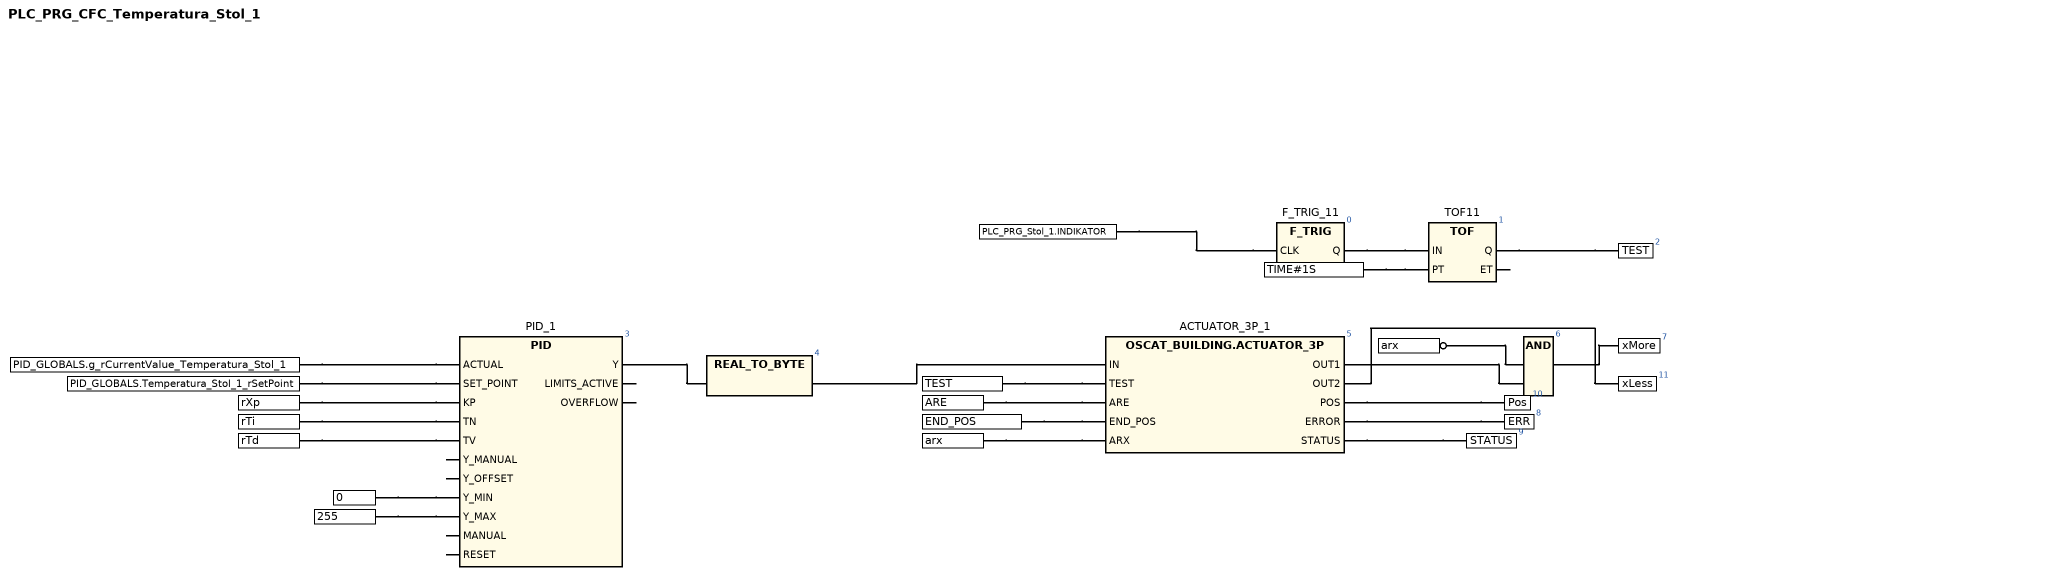
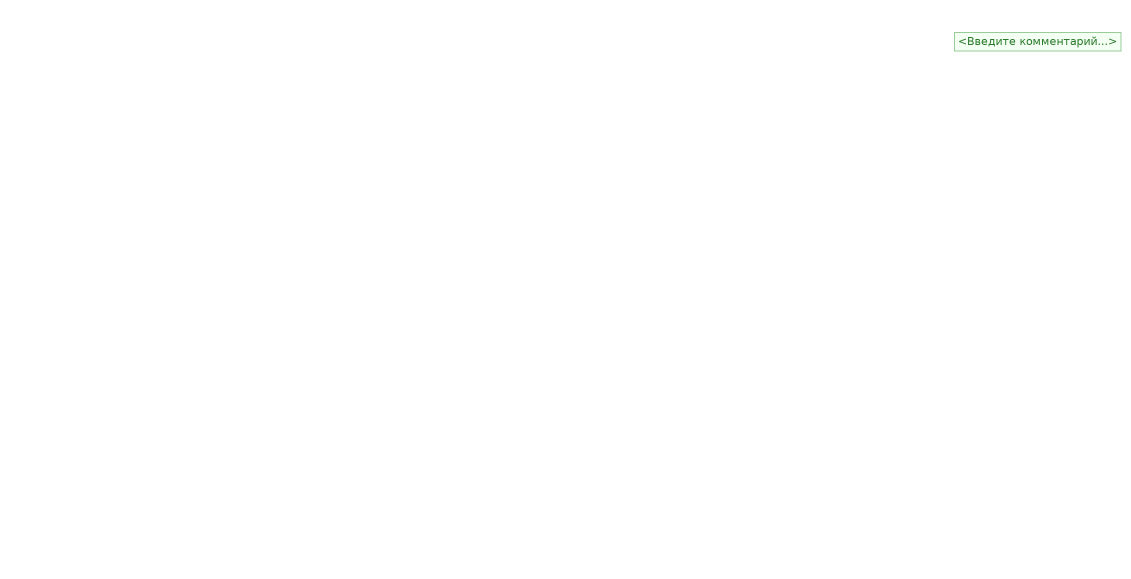
F_TRIG_11(CLK := PLC_PRG_Stol_1.INDIKATOR); // F_TRIG
TOF11(IN := F_TRIG_11.Q, PT := TIME#1S); // TOF
// <Введите комментарий...>
TEST := TOF11.Q;
PID_1(
    ACTUAL := PID_GLOBALS.g_rCurrentValue_Temperatura_Stol_1,
    SET_POINT := PID_GLOBALS.Temperatura_Stol_1_rSetPoint,
    KP := rXp,
    TN := rTi,
    TV := rTd,
    Y_MIN := 0,
    Y_MAX := 255); // PID
// parameter ACTUATOR_3P_1.SWITCH_AVAIL := FALSE
// parameter ACTUATOR_3P_1.T_DIAG := T#10d
// parameter ACTUATOR_3P_1.T_CAL := T#10m
// parameter ACTUATOR_3P_1.T_EXT := T#10s
// parameter ACTUATOR_3P_1.T_RUN := PLC_PRG_CFC_Temperatura_Stol_1.Time_RUN
ACTUATOR_3P_1(IN := REAL_TO_BYTE(PID_1.Y), TEST := TEST, ARE := ARE, END_POS := END_POS, ARX := arx); // OSCAT_BUILDING.ACTUATOR_3P
xMore := NOT arx AND ACTUATOR_3P_1.OUT1;
ERR := ACTUATOR_3P_1.ERROR;
STATUS := ACTUATOR_3P_1.STATUS;
Pos := ACTUATOR_3P_1.POS;
xLess := ACTUATOR_3P_1.OUT2;

END_PROGRAM

// Device/Application/CFC_Temperatura_PID/PLC_PRG_CFC_Temperatura_Stol_3
PROGRAM PLC_PRG_CFC_Temperatura_Stol_3
VAR
	ACTUATOR_3P_1:		OSCAT_BUILDING.ACTUATOR_3P;
	PID_1: 				PID;						// ФБ ПИД
	arx: 				BOOL;
	xMore:				BOOL;						// Сигнал открытия
	xLess: 				BOOL;						// Сигнал на закрытие	
	TEST: 				BOOL;						// Переменная запускающая тестирование ФБ ACTUATOR_3P
	Pos: 				BYTE;						// Переменная принимающая позицию 3-х ходового клапана виртуальную
	
	ARE: BOOL;
	END_POS: BOOL;
	ERR: BOOL;
	STATUS: BYTE;
	F_TRIG_21: F_TRIG;
	TOF21: TOF;
END_VAR

VAR RETAIN
	rXp: 									REAL:=2;					// Полоса пропускания (100/Кр)
	rTi: 									REAL:=25;					// Постоянная времени интегрирования
	rTd: 									REAL:=0.01;					// Постоянная времени дифференцирования
	Time_RUN:								TIME:=T#120S;				// Время хода 3-х ходового клапана
END_VAR

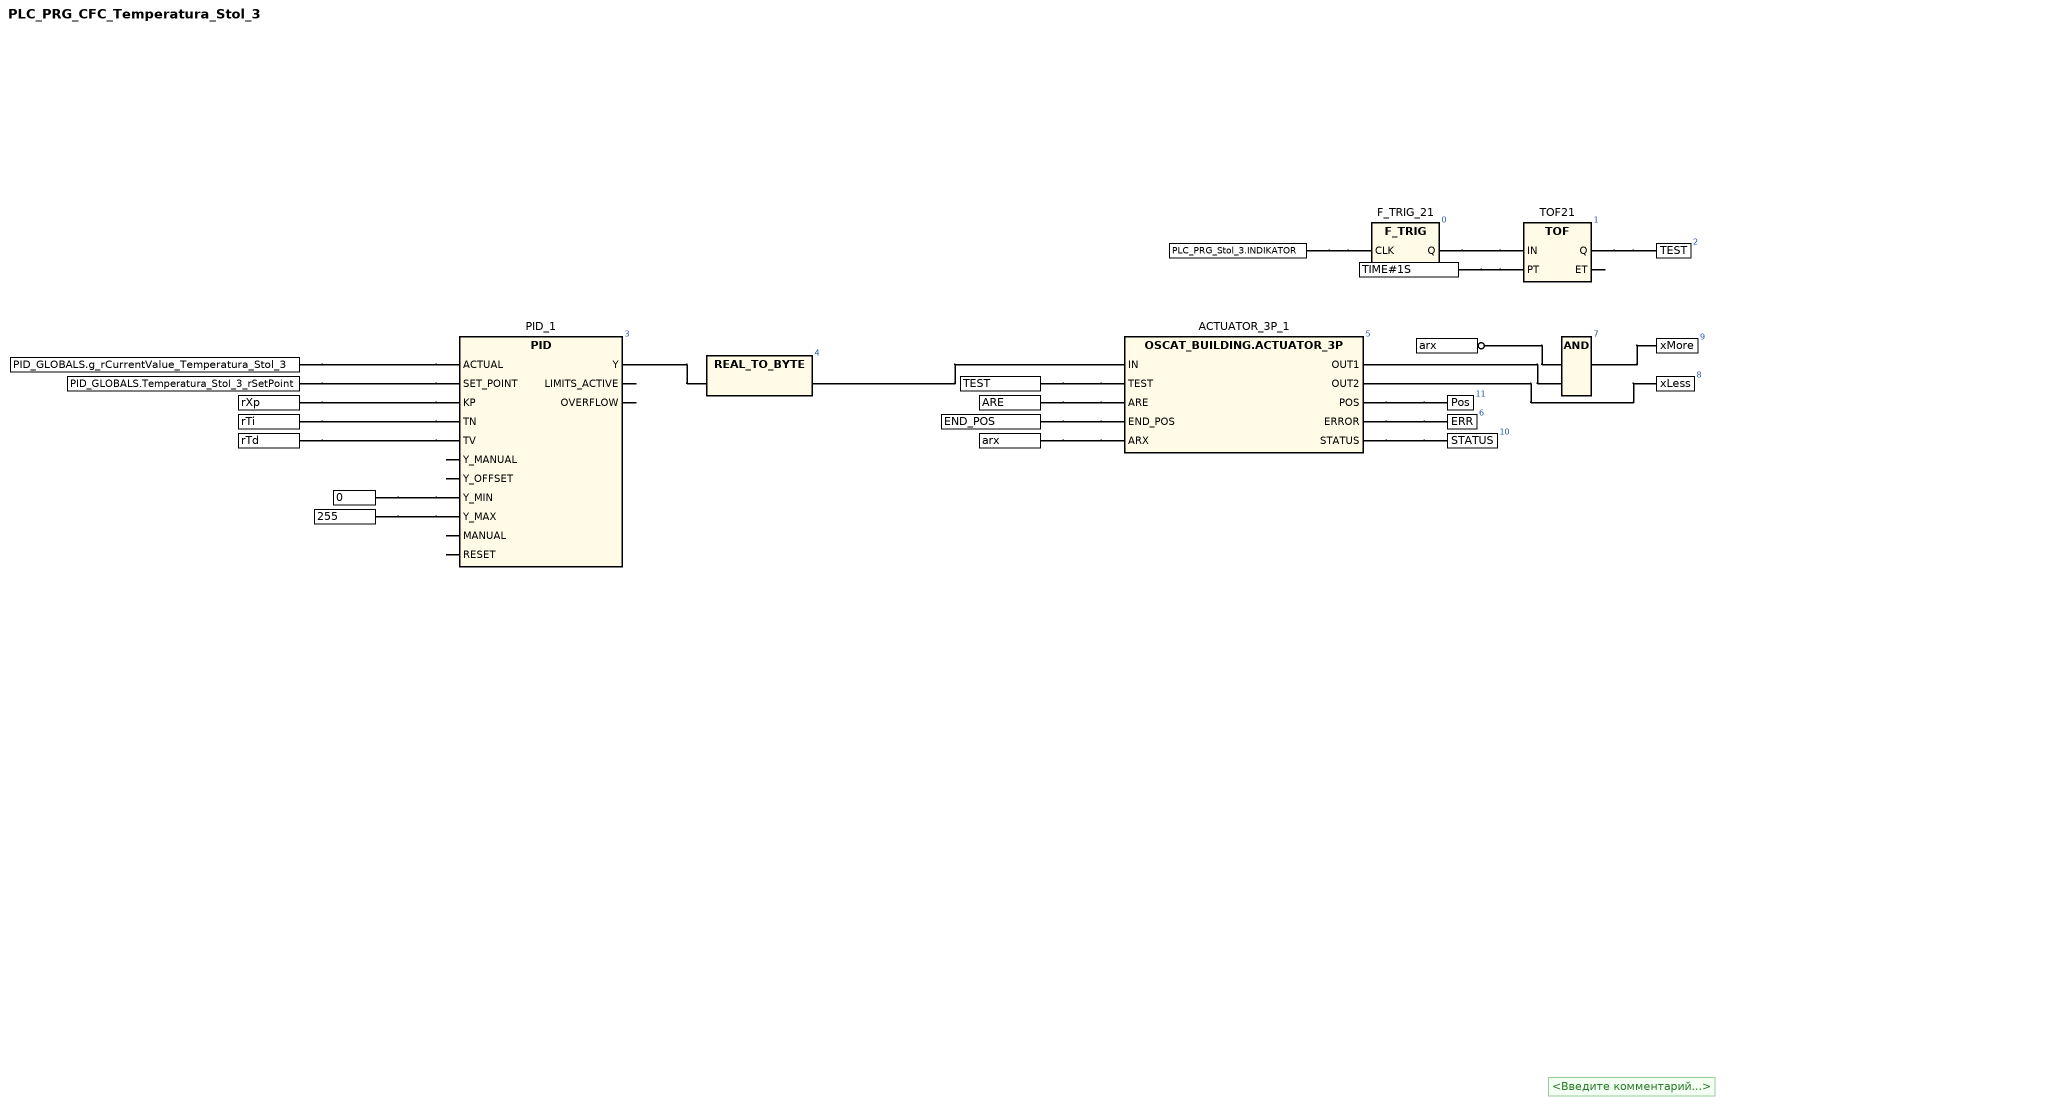
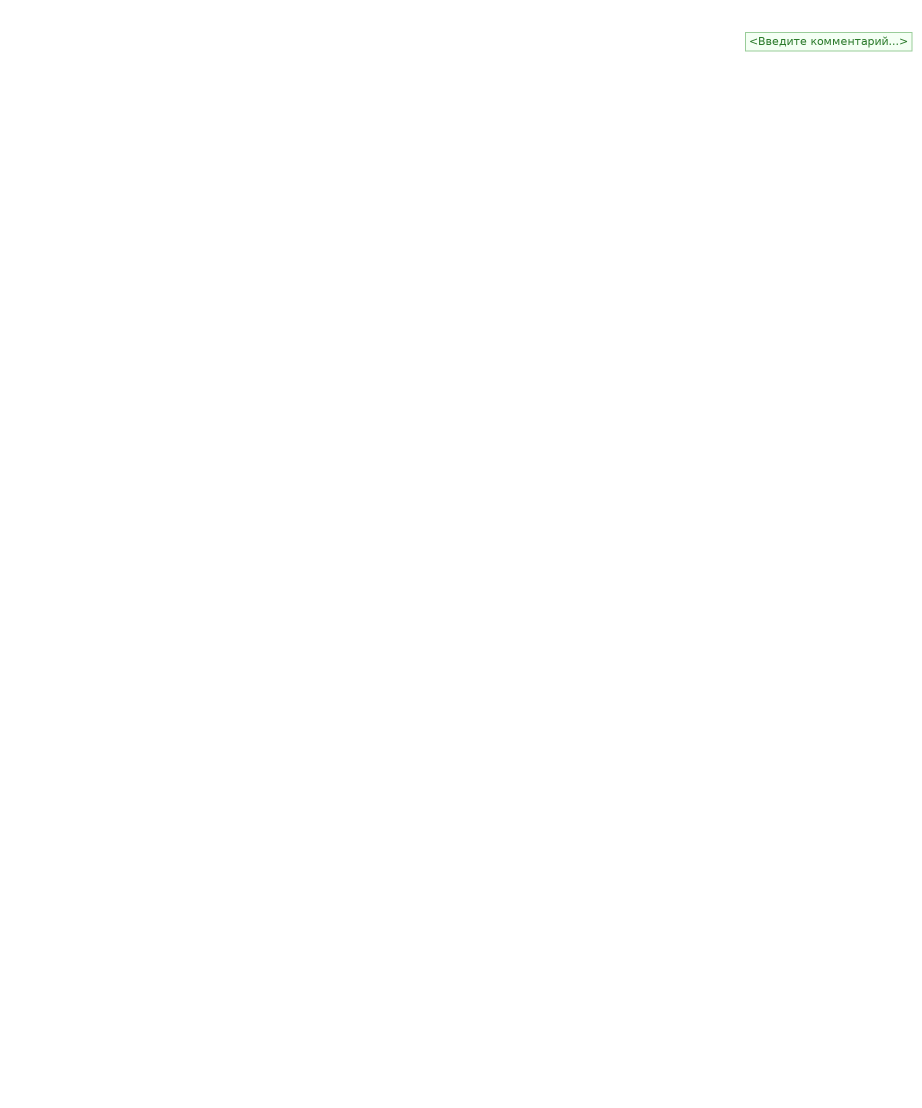
F_TRIG_21(CLK := PLC_PRG_Stol_3.INDIKATOR); // F_TRIG
TOF21(IN := F_TRIG_21.Q, PT := TIME#1S); // TOF
// <Введите комментарий...>
TEST := TOF21.Q;
PID_1(
    ACTUAL := PID_GLOBALS.g_rCurrentValue_Temperatura_Stol_3,
    SET_POINT := PID_GLOBALS.Temperatura_Stol_3_rSetPoint,
    KP := rXp,
    TN := rTi,
    TV := rTd,
    Y_MIN := 0,
    Y_MAX := 255); // PID
// parameter ACTUATOR_3P_1.SWITCH_AVAIL := FALSE
// parameter ACTUATOR_3P_1.T_DIAG := T#10d
// parameter ACTUATOR_3P_1.T_CAL := T#10m
// parameter ACTUATOR_3P_1.T_EXT := T#10s
// parameter ACTUATOR_3P_1.T_RUN := PLC_PRG_CFC_Temperatura_Stol_3.Time_RUN
ACTUATOR_3P_1(IN := REAL_TO_BYTE(PID_1.Y), TEST := TEST, ARE := ARE, END_POS := END_POS, ARX := arx); // OSCAT_BUILDING.ACTUATOR_3P
ERR := ACTUATOR_3P_1.ERROR;
xLess := ACTUATOR_3P_1.OUT2;
xMore := NOT arx AND ACTUATOR_3P_1.OUT1;
// <Введите комментарий...>
STATUS := ACTUATOR_3P_1.STATUS;
Pos := ACTUATOR_3P_1.POS;

END_PROGRAM

// Device/Application/CFC_Temperatura_PID/PLC_PRG_CFC_Temperatura_Stol_4
PROGRAM PLC_PRG_CFC_Temperatura_Stol_4
VAR
	ACTUATOR_3P_1:		OSCAT_BUILDING.ACTUATOR_3P;
	PID_1: 				PID;						// ФБ ПИД
	arx: 				BOOL;
	xMore:				BOOL;						// Сигнал открытия
	xLess: 				BOOL;						// Сигнал на закрытие
	
	TEST: 				BOOL;						// Переменная запускающая тестирование ФБ ACTUATOR_3P
	Pos: 				BYTE;						// Переменная принимающая позицию 3-х ходового клапана виртуальную
	
	ARE: BOOL;
	END_POS: BOOL;
	ERR: BOOL;
	STATUS: BYTE;
	F_TRIG_11: F_TRIG;
	TOF11: TOF;
END_VAR

VAR RETAIN	
	rXp: 									REAL:=2;					// Полоса пропускания (100/Кр)
	rTi: 									REAL:=25;					// Постоянная времени интегрирования
	rTd: 									REAL:=0.01;					// Постоянная времени дифференцирования
	Time_RUN:								TIME:=T#120S;				// Время хода 3-х ходового клапана
END_VAR

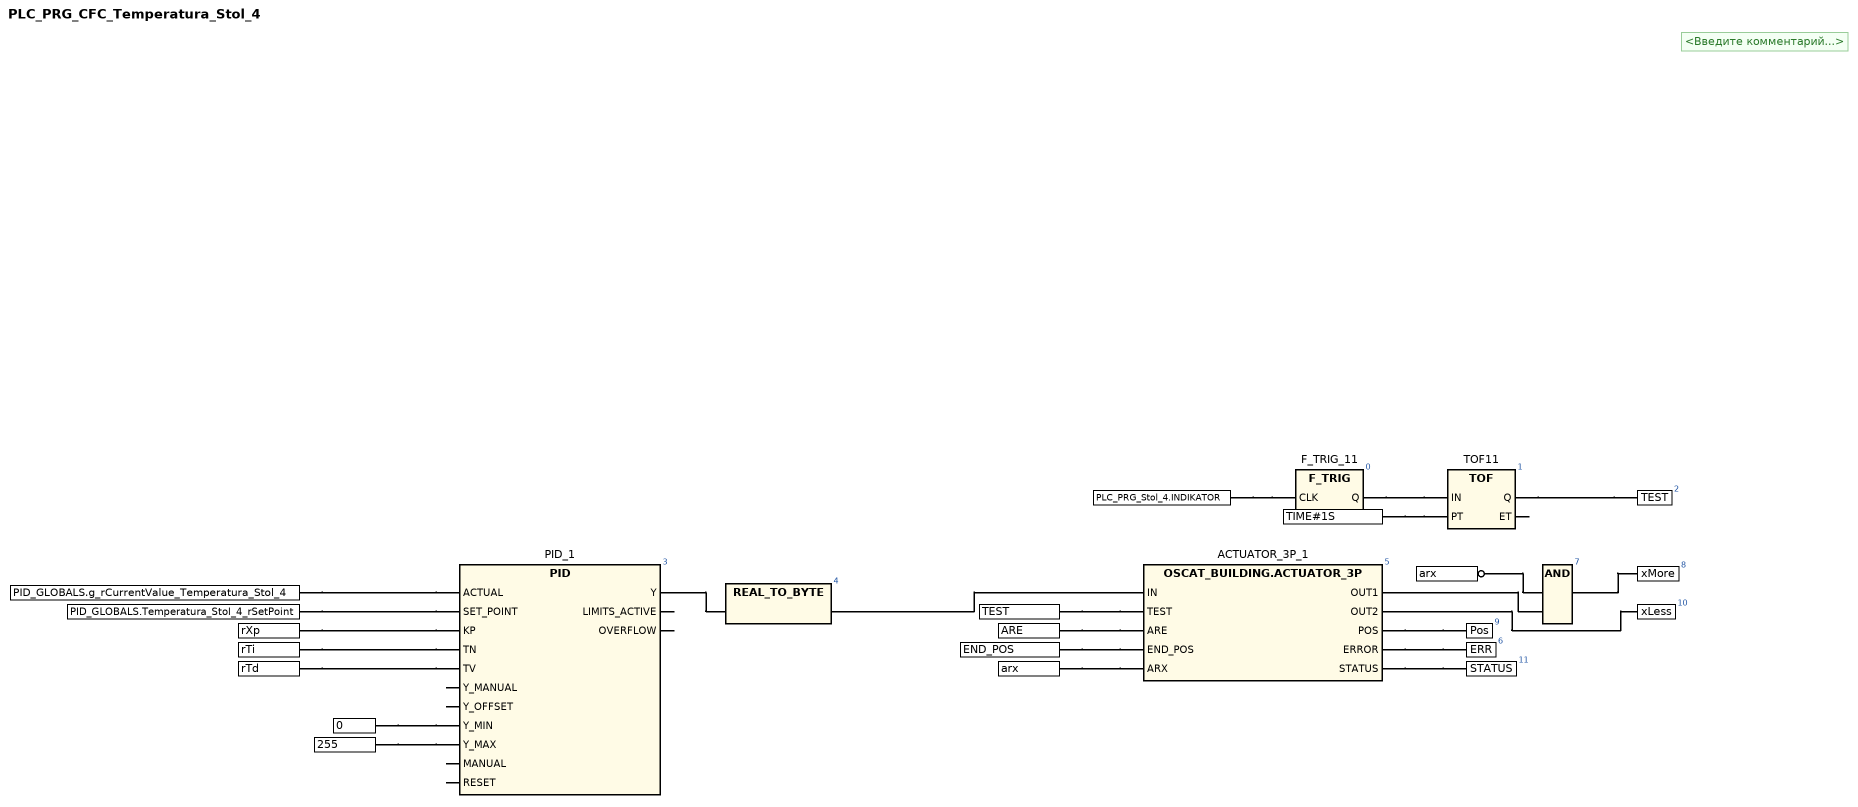
F_TRIG_11(CLK := PLC_PRG_Stol_4.INDIKATOR); // F_TRIG
TOF11(IN := F_TRIG_11.Q, PT := TIME#1S); // TOF
// <Введите комментарий...>
TEST := TOF11.Q;
PID_1(
    ACTUAL := PID_GLOBALS.g_rCurrentValue_Temperatura_Stol_4,
    SET_POINT := PID_GLOBALS.Temperatura_Stol_4_rSetPoint,
    KP := rXp,
    TN := rTi,
    TV := rTd,
    Y_MIN := 0,
    Y_MAX := 255); // PID
// parameter ACTUATOR_3P_1.SWITCH_AVAIL := FALSE
// parameter ACTUATOR_3P_1.T_DIAG := T#10d
// parameter ACTUATOR_3P_1.T_CAL := T#10m
// parameter ACTUATOR_3P_1.T_EXT := T#10s
// parameter ACTUATOR_3P_1.T_RUN := PLC_PRG_CFC_Temperatura_Stol_4.Time_RUN
ACTUATOR_3P_1(IN := REAL_TO_BYTE(PID_1.Y), TEST := TEST, ARE := ARE, END_POS := END_POS, ARX := arx); // OSCAT_BUILDING.ACTUATOR_3P
ERR := ACTUATOR_3P_1.ERROR;
xMore := NOT arx AND ACTUATOR_3P_1.OUT1;
Pos := ACTUATOR_3P_1.POS;
xLess := ACTUATOR_3P_1.OUT2;
STATUS := ACTUATOR_3P_1.STATUS;

END_PROGRAM

// Device/Application/archive/PLC_PRG_archive
PROGRAM PLC_PRG_archive
VAR
	//проверка работы архива
	//xArchEnable:				BOOL;								// бит управления архиватором
	xArchError_1:				OwenArchiverErrors.ARCHIVE_ERROR;	// код ошибки
	wsArchError_1:				WSTRING;							// сообщение об ошибке
	xArchStatus_1:				BOOL;								// статус архиватора (TRUE - запущен, FALSE - остановлен)

	// 3 и 4 стол
	xArchError_3_4:				OwenArchiverErrors.ARCHIVE_ERROR;	// код ошибки
	wsArchError_3_4:			WSTRING;							// сообщение об ошибке
	xArchStatus_3_4:			BOOL;								// статус архиватора (TRUE - запущен, FALSE - остановлен)
	
	La_rat:						BOOL;								// памяти осталось меньше 2 ГБ
	rat:						REAL;								// конвертация wstring в sint
	
	Name:						STRING;								// Имя человека активного сейчас
	
	// информация о накопителе
	xDriveInfo:					BOOL;								// режим сбора данных (TRUE - вкл.)
	
	stPlcMemory:				DriveInfo;							// структура параметров памяти контроллера
	stUsbMemory:				DriveInfo;							// структура параметров памяти USB-накопителя 
	
	fbUsbUnmountTimeout:		TON;								// таймер сброса флага "USB отмонтирован"
	
	xArchError_3_4_1:			OwenArchiverErrors.ARCHIVE_ERROR;	// статус архиватора (TRUE - запущен, FALSE - остановлен)
	warning_2:					BOOL;								// Ошибка остановлена архивация на флешку	
	warning_3:					BOOL;								// Ошибка "Неверный путь ведения архива"
	warning_4:					BOOL;								// Ошибка "Ошибка создания структуры директорий"
	warning_5:					BOOL;								// Ошибка "Ошибка удаления файла"
	warning_6:					BOOL;								// Ошибка "Ошибка переименования файла"
	warning_7:					BOOL;								// Ошибка "Некорректный буфер записи"
	warning_8:					BOOL;								// Ошибка "Некорректный размер буфера записи"
	warning_9:					BOOL;								// Ошибка "Не задан список переменных"
	warning_10:					BOOL;								// Ошибка "Список переменных пуст"
	warning_11:					BOOL;								// Ошибка "Ошибка записи"
	warning_12:					BOOL;								// Ошибка "Ошибка создания заголовка файла"
	warning_13:					BOOL;								// Ошибка "Ошибка буфер переполнен"
	
	
	x1:							BOOL;								// Отображение измененинй на 1 столе
	y1:							BOOL;								// Отображение измененинй на 3 столе
	z1:							BOOL;								// Отображение измененинй на 4 столе
	
END_VAR

// конвертируем код ошибки архиватора в строку
wsArchError_1 := OwenArchiverErrors.ARCHIVE_ERROR_TO_WSTRING(xArchError_1);

// конвертируем код ошибки архиватора в строку
wsArchError_3_4 := OwenArchiverErrors.ARCHIVE_ERROR_TO_WSTRING(xArchError_3_4);

act01_DriveInfo();			// сбор информации о памяти накомпителя и ПЛК

rat := WSTRING_TO_SINT(stUsbMemory.wsFreeSize);

IF rat > 2  THEN				// поменять цифру 2 на 4 когда придёт флешка
	La_rat  := TRUE;			// надо почистить флешку на термостолах
END_IF

// Проверка записи архива на флешку
IF xArchStatus_1 = TRUE OR xArchStatus_3_4 = TRUE THEN
	warning_2 := TRUE;
ELSE
	warning_2 := FALSE;
END_IF

Name := TO_STRING(VisuElems.CurrentFullUserName);


// Определение последней ошибки архивации
IF xArchError_3_4_1 = ARCHIVE_ERROR.INCORRECT_ARCHIVE_PATH THEN
	warning_3 := TRUE;
	warning_4 := FALSE;
	warning_5 := FALSE;
	warning_6 := FALSE;
	warning_7 := FALSE;
	warning_8 := FALSE;
	warning_9 := FALSE;
	warning_10 := FALSE;
	warning_11 := FALSE;
	warning_12 := FALSE;
	warning_13 := FALSE;
	ELSIF xArchError_3_4_1 = ARCHIVE_ERROR.CREATE_FOLDER_STRUCTURE_ERROR THEN
	warning_4 := TRUE;
	warning_3 := FALSE;
	warning_5 := FALSE;
	warning_6 := FALSE;
	warning_7 := FALSE;
	warning_8 := FALSE;
	warning_9 := FALSE;
	warning_10 := FALSE;
	warning_11 := FALSE;
	warning_12 := FALSE;
	warning_13 := FALSE;
	ELSIF xArchError_3_4_1 = ARCHIVE_ERROR.DELETE_FILE_ERROR THEN
	warning_5 := TRUE;
	warning_3 := FALSE;
	warning_4 := FALSE;
	warning_6 := FALSE;
	warning_7 := FALSE;
	warning_8 := FALSE;
	warning_9 := FALSE;
	warning_10 := FALSE;
	warning_11 := FALSE;
	warning_12 := FALSE;
	warning_13 := FALSE;
	ELSIF xArchError_3_4_1 = ARCHIVE_ERROR.RENAME_FILE_ERROR THEN
	warning_3 := FALSE;
	warning_4 := FALSE;
	warning_5 := FALSE;
	warning_6 := TRUE;
	warning_7 := FALSE;
	warning_8 := FALSE;
	warning_9 := FALSE;
	warning_10 := FALSE;
	warning_11 := FALSE;
	warning_12 := FALSE;
	warning_13 := FALSE;
	ELSIF xArchError_3_4_1 = ARCHIVE_ERROR.INCORRECT_WRITER_BUFFER THEN
	warning_3 := FALSE;
	warning_4 := FALSE;
	warning_5 := FALSE;
	warning_6 := FALSE;
	warning_7 := TRUE;
	warning_8 := FALSE;
	warning_9 := FALSE;
	warning_10 := FALSE;
	warning_11 := FALSE;
	warning_12 := FALSE;
	warning_13 := FALSE;
	ELSIF xArchError_3_4_1 = ARCHIVE_ERROR.INCORRECT_WRITER_BUFFER_SIZE THEN
	warning_3 := FALSE;
	warning_4 := FALSE;
	warning_5 := FALSE;
	warning_6 := FALSE;
	warning_7 := FALSE;
	warning_8 := TRUE;
	warning_9 := FALSE;
	warning_10 := FALSE;
	warning_11 := FALSE;
	warning_12 := FALSE;
	warning_13 := FALSE;
	ELSIF xArchError_3_4_1 = ARCHIVE_ERROR.VARIABLE_LIST_NOT_SPECIFIED THEN
	warning_3 := FALSE;
	warning_4 := FALSE;
	warning_5 := FALSE;
	warning_6 := FALSE;
	warning_7 := FALSE;
	warning_8 := FALSE;
	warning_9 := TRUE;
	warning_10 := FALSE;
	warning_11 := FALSE;
	warning_12 := FALSE;
	warning_13 := FALSE;
	ELSIF xArchError_3_4_1 = ARCHIVE_ERROR.VARIABLE_LIST_IS_EMPTY THEN
	warning_3 := FALSE;
	warning_4 := FALSE;
	warning_5 := FALSE;
	warning_6 := FALSE;
	warning_7 := FALSE;
	warning_8 := FALSE;
	warning_9 := FALSE;
	warning_10 := TRUE;
	warning_11 := FALSE;
	warning_12 := FALSE;
	warning_13 := FALSE;
	ELSIF xArchError_3_4_1 = ARCHIVE_ERROR.WRITE_ERROR THEN
	warning_3 := FALSE;
	warning_4 := FALSE;
	warning_5 := FALSE;
	warning_6 := FALSE;
	warning_7 := FALSE;
	warning_8 := FALSE;
	warning_9 := FALSE;
	warning_10 := FALSE;
	warning_11 := TRUE;
	warning_12 := FALSE;
	warning_13 := FALSE;
	ELSIF xArchError_3_4_1 = ARCHIVE_ERROR.CREATE_HEADER_ERROR THEN
	warning_3 := FALSE;
	warning_4 := FALSE;
	warning_5 := FALSE;
	warning_6 := FALSE;
	warning_7 := FALSE;
	warning_8 := FALSE;
	warning_9 := FALSE;
	warning_10 := FALSE;
	warning_11 := FALSE;
	warning_12 := TRUE;
	warning_13 := FALSE;
	ELSIF xArchError_3_4_1 = ARCHIVE_ERROR.WRITE_BUFFER_OVERFLOW THEN
	warning_3 := FALSE;
	warning_4 := FALSE;
	warning_5 := FALSE;
	warning_6 := FALSE;
	warning_7 := FALSE;
	warning_8 := FALSE;
	warning_9 := FALSE;
	warning_10 := FALSE;
	warning_11 := FALSE;
	warning_12 := FALSE;
	warning_13 := TRUE;
	ELSE
	warning_3 := FALSE;
	warning_4 := FALSE;
	warning_5 := FALSE;
	warning_6 := FALSE;
	warning_7 := FALSE;
	warning_8 := FALSE;
	warning_9 := FALSE;
	warning_10 := FALSE;
	warning_11 := FALSE;
	warning_12 := FALSE;
	warning_13 := FALSE;
END_IF

ACTION act01_DriveInfo:
// преобразование размеров полной/занятой/свободной памяти в форматированную строку

stPlcMemory.wsFullSize 		:= BYTE_SIZE_TO_WSTRING(stPlcMemory.uleFullSize);
stPlcMemory.wsUsedSize 		:= BYTE_SIZE_TO_WSTRING(stPlcMemory.uleUsedSize);
stPlcMemory.wsFreeSize 		:= BYTE_SIZE_TO_WSTRING(stPlcMemory.uleFreeSize);

stUsbMemory.wsFullSize 		:= BYTE_SIZE_TO_WSTRING(stUsbMemory.uleFullSize);
stUsbMemory.wsUsedSize 		:= BYTE_SIZE_TO_WSTRING(stUsbMemory.uleUsedSize);
stUsbMemory.wsFreeSize 		:= BYTE_SIZE_TO_WSTRING(stUsbMemory.uleFreeSize);

// сброс флагов "устройство отмонтировано" через 5 секунд после отмонтирования устройства
fbUsbUnmountTimeout(IN:=stUsbMemory.xUnmountDone, PT:=T#5S);

IF fbUsbUnmountTimeout.Q THEN
	stUsbMemory.xUnmount:=FALSE;
END_IF
END_ACTION

END_PROGRAM

// Device/Application/archive/BYTE_SIZE_TO_WSTRING
// функция преобразования числа байт в форматированную строку
FUNCTION BYTE_SIZE_TO_WSTRING : WSTRING
VAR_INPUT
	uliByteSize: 				ULINT; 				// число байт
END_VAR
VAR CONSTANT
	c_uliBytePerKilobyte: 		ULINT := 1024; 		// число байт в килобайте
	c_uliKilobytePerMegabyte: 	ULINT := 1024 * c_uliBytePerKilobyte;
	c_uliMegabytePerGigabyte: 	ULINT := 1024 * c_uliKilobytePerMegabyte;
END_VAR
VAR
	rByteSize: 					REAL; 				// промежуточная переменная
END_VAR

CASE uliByteSize OF
	

	0 ..(c_uliBytePerKilobyte - 1):
			BYTE_SIZE_TO_WSTRING := WCONCAT(ULINT_TO_WSTRING(uliByteSize), " Байт");

	c_uliBytePerKilobyte ..(c_uliKilobytePerMegabyte - 1):
			rByteSize := ULINT_TO_REAL(uliByteSize) / ULINT_TO_REAL(c_uliBytePerKilobyte);
			BYTE_SIZE_TO_WSTRING := WCONCAT(REAL_TO_FWSTRING(rByteSize, 2), " Кбайт");

	c_uliKilobytePerMegabyte ..(c_uliMegabytePerGigabyte - 1):
			rByteSize := ULINT_TO_REAL(uliByteSize) / ULINT_TO_REAL(c_uliKilobytePerMegabyte);
			BYTE_SIZE_TO_WSTRING := WCONCAT(REAL_TO_FWSTRING(rByteSize, 2), " Мбайт");

	c_uliMegabytePerGigabyte ..(32 * c_uliMegabytePerGigabyte):
			rByteSize := ULINT_TO_REAL(uliByteSize) / ULINT_TO_REAL(c_uliMegabytePerGigabyte);
			BYTE_SIZE_TO_WSTRING := WCONCAT(REAL_TO_FWSTRING(rByteSize, 2), " Гбайт");
			
END_CASE

END_FUNCTION

// Device/Application/archive/REAL_TO_FWSTRING
// функция конвертирует значение типа REAL в строку с n знаков после запятой
FUNCTION REAL_TO_FWSTRING : WSTRING

VAR_INPUT
	rVar: 			REAL; 		// входное значение
	usiPrecision: 	USINT; 		// нужное кол-во знаков после запятой
END_VAR
VAR
	uliVar: 		ULINT; 		// промежуточная переменная
	lrVar: 			LREAL; 		// промежуточная переменная
END_VAR



uliVar := LREAL_TO_ULINT( (rVar)*EXPT(10, usiPrecision) );
lrVar := LINT_TO_LREAL(uliVar) / EXPT(10, usiPrecision);
REAL_TO_FWSTRING := LREAL_TO_WSTRING(lrVar);

END_FUNCTION

// Device/Application/Connection
PROGRAM Connection
VAR
	// Модуль расширения MK210_311_Stol_1_2
	sName_MK210_311_Stol_1_2:					STRING;						// Имя модуля, считанное с модуля
	sProjectName_MK210_311_Stol_1_2:			STRING;						// Имя модуля в дереве проекта
	abyIP_MK210_311_Stol_1_2:					ARRAY [0..3] OF BYTE;		// IP-адрес в дереве проекта
	sFactoryNumber_MK210_311_Stol_1_2:			STRING;						// заводской номер модуля
	udiErrorsCount_MK210_311_Stol_1_2:			UDINT;						// Число ошибок связи с модулем с последней загрузки контроллера
	eLastError_MK210_311_Stol_1_2: 				MB_ERRORCODES;				// код последней ошибки
	ePollState_MK210_311_Stol_1_2:				MODULE_STATE;				// состояние опроса
	
	// Модуль расширения MV210_212_Stol_1_2
	sName_MV210_212_Stol_1_2:					STRING;						// Имя модуля, считанное с модуля
	sProjectName_MV210_212_Stol_1_2:			STRING;						// Имя модуля в дереве проекта
	abyIP_MV210_212_Stol_1_2:					ARRAY [0..3] OF BYTE;		// IP-адрес в дереве проекта
	sFactoryNumber_MV210_212_Stol_1_2:			STRING;						// заводской номер модуля
	udiErrorsCount_MV210_212_Stol_1_2:			UDINT;						// Число ошибок связи с модулем с последней загрузки контроллера
	eLastError_MV210_212_Stol_1_2: 				MB_ERRORCODES;				// код последней ошибки
	ePollState_MV210_212_Stol_1_2:				MODULE_STATE;				// состояние опроса
	
	// Модуль расширения MV210_101_Stol_1_2
	sName_MV210_101_Stol_1_2:					STRING;						// Имя модуля, считанное с модуля
	sProjectName_MV210_101_Stol_1_2:			STRING;						// Имя модуля в дереве проекта
	abyIP_MV210_101_Stol_1_2:					ARRAY [0..3] OF BYTE;		// IP-адрес в дереве проекта
	sFactoryNumber_MV210_101_Stol_1_2:			STRING;						// заводской номер модуля
	udiErrorsCount_MV210_101_Stol_1_2:			UDINT;						// Число ошибок связи с модулем с последней загрузки контроллера
	eLastError_MV210_101_Stol_1_2: 				MB_ERRORCODES;				// код последней ошибки
	ePollState_MV210_101_Stol_1_2:				MODULE_STATE;				// состояние опроса
	
	// Модуль расширения MK210_311_Stol_3_4
	sName_MK210_311_Stol_3_4:					STRING;						// Имя модуля, считанное с модуля
	sProjectName_MK210_311_Stol_3_4:			STRING;						// Имя модуля в дереве проекта
	abyIP_MK210_311_Stol_3_4:					ARRAY [0..3] OF BYTE;		// IP-адрес в дереве проекта
	sFactoryNumber_MK210_311_Stol_3_4:			STRING;						// заводской номер модуля
	udiErrorsCount_MK210_311_Stol_3_4:			UDINT;						// Число ошибок связи с модулем с последней загрузки контроллера
	eLastError_MK210_311_Stol_3_4: 				MB_ERRORCODES;				// код последней ошибки
	ePollState_MK210_311_Stol_3_4:				MODULE_STATE;				// состояние опроса
	
	// Модуль расширения MV210_212_Stol_3_4
	sName_MV210_212_Stol_3_4:					STRING;						// Имя модуля, считанное с модуля
	sProjectName_MV210_212_Stol_3_4:			STRING;						// Имя модуля в дереве проекта
	abyIP_MV210_212_Stol_3_4:					ARRAY [0..3] OF BYTE;		// IP-адрес в дереве проекта
	sFactoryNumber_MV210_212_Stol_3_4:			STRING;						// заводской номер модуля
	udiErrorsCount_MV210_212_Stol_3_4:			UDINT;						// Число ошибок связи с модулем с последней загрузки контроллера
	eLastError_MV210_212_Stol_3_4: 				MB_ERRORCODES;				// код последней ошибки
	ePollState_MV210_212_Stol_3_4:				MODULE_STATE;				// состояние опроса
	
	// Модуль расширения MV210_101_Stol_3_4
	sName_MV210_101_Stol_3_4:					STRING;						// Имя модуля, считанное с модуля
	sProjectName_MV210_101_Stol_3_4:			STRING;						// Имя модуля в дереве проекта
	abyIP_MV210_101_Stol_3_4:					ARRAY [0..3] OF BYTE;		// IP-адрес в дереве проекта
	sFactoryNumber_MV210_101_Stol_3_4:			STRING;						// Pаводской номер модуля
	udiErrorsCount_MV210_101_Stol_3_4:			UDINT;						// Число ошибок связи с модулем с последней загрузки контроллера
	eLastError_MV210_101_Stol_3_4: 				MB_ERRORCODES;				// Rод последней ошибки
	ePollState_MV210_101_Stol_3_4:				MODULE_STATE;				// Cостояние опроса
		
	warning:									BOOL;						// Ошибка модулей расширения 1 стола
	warning_1:									BOOL;						// Ошибка модулей расширения 3 и 4 столов
END_VAR

// Модуль расширения MK210_311_Stol_1_2
sName_MK210_311_Stol_1_2				:=  MK210_311_Stol_1_2_OwenDriver.Name;
sProjectName_MK210_311_Stol_1_2			:=	MK210_311_Stol_1_2_OwenDriver.ProjectName;
abyIP_MK210_311_Stol_1_2				:=	MK210_311_Stol_1_2_OwenDriver.Ip;
sFactoryNumber_MK210_311_Stol_1_2 		:=	MK210_311_Stol_1_2_OwenDriver.FactoryNumber;
udiErrorsCount_MK210_311_Stol_1_2		:=	MK210_311_Stol_1_2_OwenDriver.ErrorsCount;
eLastError_MK210_311_Stol_1_2 			:=	MK210_311_Stol_1_2_OwenDriver.LastError;
ePollState_MK210_311_Stol_1_2			:=	MK210_311_Stol_1_2_OwenDriver.PollState;

// Модуль расширения MV210_212_Stol_1_2
sName_MV210_212_Stol_1_2				:=  MV210_212_Stol_1_2_OwenDriver.Name;
sProjectName_MV210_212_Stol_1_2			:=	MV210_212_Stol_1_2_OwenDriver.ProjectName;
abyIP_MV210_212_Stol_1_2				:=	MV210_212_Stol_1_2_OwenDriver.Ip;
sFactoryNumber_MV210_212_Stol_1_2 		:=	MV210_212_Stol_1_2_OwenDriver.FactoryNumber;
udiErrorsCount_MV210_212_Stol_1_2		:=	MV210_212_Stol_1_2_OwenDriver.ErrorsCount;
eLastError_MV210_212_Stol_1_2 			:=	MV210_212_Stol_1_2_OwenDriver.LastError;
ePollState_MV210_212_Stol_1_2			:=	MV210_212_Stol_1_2_OwenDriver.PollState;

// Модуль расширения MV210_101_Stol_1_2
sName_MV210_101_Stol_1_2				:=  MV210_101_Stol_1_2_OwenDriver.Name;
sProjectName_MV210_101_Stol_1_2			:=	MV210_101_Stol_1_2_OwenDriver.ProjectName;
abyIP_MV210_101_Stol_1_2				:=	MV210_101_Stol_1_2_OwenDriver.Ip;
sFactoryNumber_MV210_101_Stol_1_2	 	:=	MV210_101_Stol_1_2_OwenDriver.FactoryNumber;
udiErrorsCount_MV210_101_Stol_1_2		:=	MV210_101_Stol_1_2_OwenDriver.ErrorsCount;
eLastError_MV210_101_Stol_1_2 			:=	MV210_101_Stol_1_2_OwenDriver.LastError;
ePollState_MV210_101_Stol_1_2			:=	MV210_101_Stol_1_2_OwenDriver.PollState;

// Модуль расширения MK210_311_Stol_3_4
sName_MK210_311_Stol_3_4				:=  MK210_311_Stol_3_4_OwenDriver.Name;
sProjectName_MK210_311_Stol_3_4			:=	MK210_311_Stol_3_4_OwenDriver.ProjectName;
abyIP_MK210_311_Stol_3_4				:=	MK210_311_Stol_3_4_OwenDriver.Ip;
sFactoryNumber_MK210_311_Stol_3_4 		:=	MK210_311_Stol_3_4_OwenDriver.FactoryNumber;
udiErrorsCount_MK210_311_Stol_3_4		:=	MK210_311_Stol_3_4_OwenDriver.ErrorsCount;
eLastError_MK210_311_Stol_3_4 			:=	MK210_311_Stol_3_4_OwenDriver.LastError;
ePollState_MK210_311_Stol_3_4			:=	MK210_311_Stol_3_4_OwenDriver.PollState;

// Модуль расширения MV210_212_Stol_3_4
sName_MV210_212_Stol_3_4				:=  MV210_212_Stol_3_4_OwenDriver.Name;
sProjectName_MV210_212_Stol_3_4			:=	MV210_212_Stol_3_4_OwenDriver.ProjectName;
abyIP_MV210_212_Stol_3_4				:=	MV210_212_Stol_3_4_OwenDriver.Ip;
sFactoryNumber_MV210_212_Stol_3_4 		:=	MV210_212_Stol_3_4_OwenDriver.FactoryNumber;
udiErrorsCount_MV210_212_Stol_3_4		:=	MV210_212_Stol_3_4_OwenDriver.ErrorsCount;
eLastError_MV210_212_Stol_3_4 			:=	MV210_212_Stol_3_4_OwenDriver.LastError;
ePollState_MV210_212_Stol_3_4			:=	MV210_212_Stol_3_4_OwenDriver.PollState;

// Модуль расширения MV210_101_Stol_3_4
sName_MV210_101_Stol_3_4				:=  MV210_101_Stol_3_4_OwenDriver.Name;
sProjectName_MV210_101_Stol_3_4			:=	MV210_101_Stol_3_4_OwenDriver.ProjectName;
abyIP_MV210_101_Stol_3_4				:=	MV210_101_Stol_3_4_OwenDriver.Ip;
sFactoryNumber_MV210_101_Stol_3_4 		:=	MV210_101_Stol_3_4_OwenDriver.FactoryNumber;
udiErrorsCount_MV210_101_Stol_3_4		:=	MV210_101_Stol_3_4_OwenDriver.ErrorsCount;
eLastError_MV210_101_Stol_3_4 			:=	MV210_101_Stol_3_4_OwenDriver.LastError;
ePollState_MV210_101_Stol_3_4			:=	MV210_101_Stol_3_4_OwenDriver.PollState;


IF ePollState_MV210_101_Stol_1_2 = MODULE_STATE.OK AND ePollState_MK210_311_Stol_1_2 = MODULE_STATE.OK  AND ePollState_MV210_212_Stol_1_2 = MODULE_STATE.OK THEN
	warning := TRUE;
ELSE
	warning := FALSE;
END_IF



IF ePollState_MV210_101_Stol_3_4 = MODULE_STATE.OK AND ePollState_MK210_311_Stol_3_4 = MODULE_STATE.OK  AND ePollState_MV210_212_Stol_3_4 = MODULE_STATE.OK THEN
	warning_1 := TRUE;
ELSE
	warning_1 := FALSE;
END_IF

END_PROGRAM

// POU_LIN_TRAFO
FUNCTION_BLOCK POU_LIN_TRAFO
VAR_INPUT
	X: REAL;
	I_LO: REAL;
	I_HI: REAL;
	O_LO: REAL;
	O_HI: REAL;
END_VAR
VAR_OUTPUT
	SCALE_B: REAL;
END_VAR

IF I_HI = I_LO THEN
	SCALE_B := O_LO;
ELSE
	SCALE_B :=(O_HI-O_LO)*((X-I_LO)/(I_HI-I_LO))+O_LO;
END_IF

END_FUNCTION_BLOCK

// Device/Application/CFC_Temperatura_PID/PLC_PRG_CFC_Temperatura_Stol_2
PROGRAM PLC_PRG_CFC_Temperatura_Stol_2
VAR
	ACTUATOR_3P_1:		OSCAT_BUILDING.ACTUATOR_3P;
	PID_1: 				PID;						// ФБ ПИД
	arx: 				BOOL;
	xMore:				BOOL;						// Сигнал открытия
	xLess: 				BOOL;						// Сигнал на закрытие
END_VAR
VAR RETAIN
	
	rXp: 									REAL:=10;					// Полоса пропускания (100/Кр)
	rTi: 									REAL:=5;					// Постоянная времени интегрирования
	rTd: 									REAL:=1;					// Постоянная времени дифференцирования
	
END_VAR

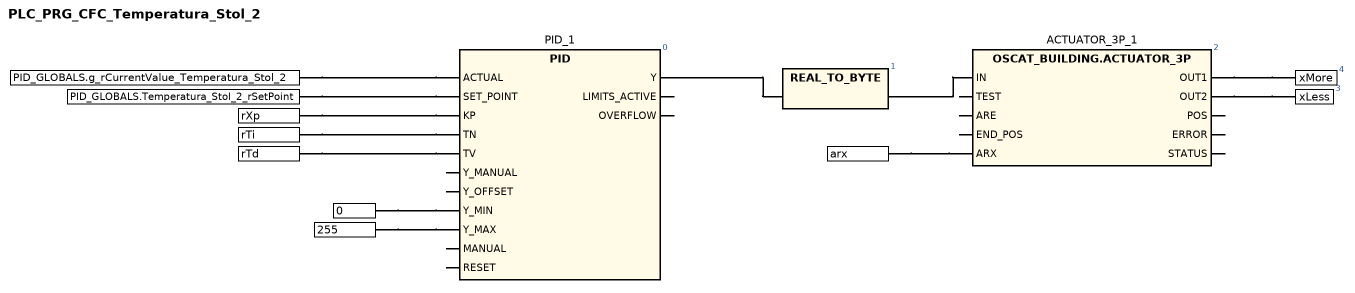
PID_1(
    ACTUAL := PID_GLOBALS.g_rCurrentValue_Temperatura_Stol_2,
    SET_POINT := PID_GLOBALS.Temperatura_Stol_2_rSetPoint,
    KP := rXp,
    TN := rTi,
    TV := rTd,
    Y_MIN := 0,
    Y_MAX := 255); // PID
ACTUATOR_3P_1(IN := REAL_TO_BYTE(PID_1.Y), ARX := arx); // OSCAT_BUILDING.ACTUATOR_3P
xLess := ACTUATOR_3P_1.OUT2;
xMore := ACTUATOR_3P_1.OUT1;

END_PROGRAM

// Device/Application/Parostol_Zadanie/Zadanie_1
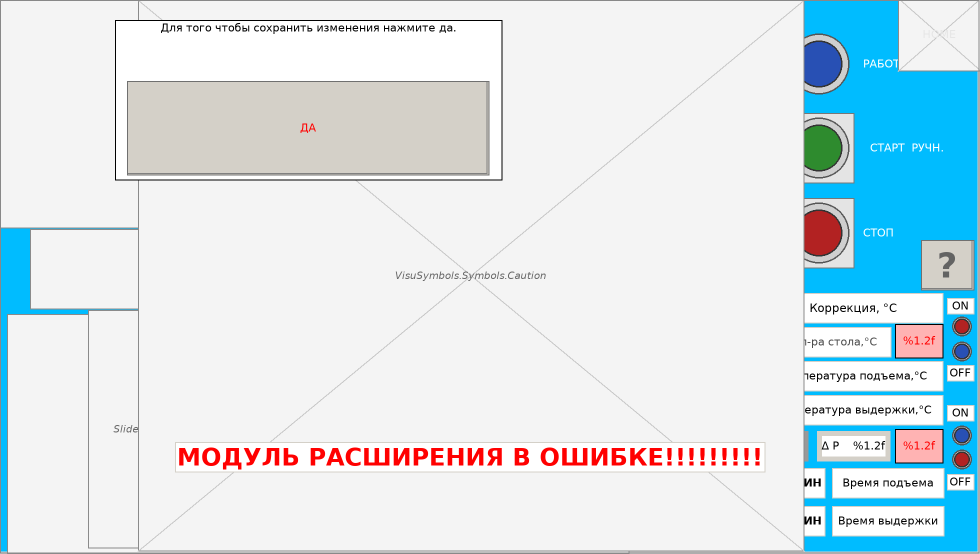
VISUALIZATION Zadanie_1  // 980x554
VAR_IN_OUT
END_VAR
VAR
	bResetTrigger : BOOL;
	bStart : BOOL;
	bStop : BOOL;
	bStore : BOOL;
	sStoreFilename : STRING;
	bRestore : BOOL;
	sRestoreFilename : STRING;
END_VAR
    Rectangle (-3,-3 980x554)
    Histogram (7,314 622x240), scale format: %.1f, scale 0..100
        p518627256: °C
        p1518820177: PLC_PRG_Stol_1.arrHist1
        p102497268: PLC_PRG.arrHist1
        p788070771: ARRAY [0..3] OF REAL
    Slider (88,310 80x238), variable: PLC_PRG_Stol_1.Y1, scale 0..100
        OnValueChanged: execute { PLC_PRG_archive.x1 := TRUE; }
    Slider (215,310 80x238), variable: PLC_PRG_Stol_1.Y2, scale 0..100
        OnValueChanged: execute { PLC_PRG_archive.x1 := TRUE; }
    Slider (354,310 80x238), variable: PLC_PRG_Stol_1.Y3, scale 0..100
        OnValueChanged: execute { PLC_PRG_archive.x1 := TRUE; }
    Slider (487,310 80x238), variable: PLC_PRG_Stol_1.Y4, scale 0..100
    Trend (-3,-2 543x230)
        p758368661: dd.MM.yyyy
        p2423372160: H:mm:ss
        p2833066001: Visualization_Trend_Stol_1
        p2059293862: GenElemInst_240
    Line (925,485)
    Textfield (648,293 108x30)
        OnMouseClick: write the text variable via Default
    Textfield (648,395 108x30), "%d", text variable: PLC_PRG_Stol_1.Y3
        OnValueChanged: execute { PLC_PRG_archive.x1 := TRUE; }
        OnMouseClick: write the text variable via Default, min 0, max 100
    Textfield (648,327 108x30), "%d", text variable: PLC_PRG_Stol_1.Y1
        OnValueChanged: execute { PLC_PRG_archive.x1 := TRUE; }
        OnMouseClick: write the text variable via Default, min 0, max 100
    Textfield (649,468 50x30), "%d", text variable: PLC_PRG_Stol_1.HX2
        OnValueChanged: execute { PLC_PRG_archive.x1 := TRUE; }
        OnMouseClick: write the text variable via Default, min 0
    Textfield (764,293 179x30), "Коррекция, °C"
    Textfield (764,327 127x30), "Темп-ра стола,°C"
    Textfield (764,361 179x30), "Температура подъема,°C"
    Textfield (764,395 179x30), "Температура выдержки,°C"
    Textfield (832,468 112x30), "Время подъема"
    Textfield (649,507 50x30), "%d", text variable: PLC_PRG_Stol_1.HX3
        OnValueChanged: execute { PLC_PRG_archive.x1 := TRUE; }
        OnMouseClick: write the text variable via Default, min 0
    Textfield (832,506 112x30), "Время выдержки"
    Textfield (167,16 150x30), "%d °C, уставка", text variable: PID_GLOBALS.Temperatura_Stol_1_rSetPoint
    Textfield (734,468 50x30), "%d", text variable: PLC_PRG_Stol_1.MX2
        OnValueChanged: execute { PLC_PRG_archive.x1 := TRUE; }
        OnMouseClick: write the text variable via Default, min 0, max 59
    Textfield (704,468 25x30), "Ч"
    Textfield (789,468 36x30), "МИН"
    Textfield (734,507 50x30), "%d", text variable: PLC_PRG_Stol_1.MX3
        OnValueChanged: execute { PLC_PRG_archive.x1 := TRUE; }
        OnMouseClick: write the text variable via Default, min 0, max 59
    Textfield (704,507 25x30), "Ч"
    Textfield (789,506 36x30), "МИН"
    Checkbox (653,36 113x35), "Понедельник", variable: NVI_RETAIN.dateWeekStolOneTwo.1
        OnValueChanged: execute { PLC_PRG_archive.x1 := TRUE; }
    Checkbox (653,71 113x35), "Вторник", variable: NVI_RETAIN.dateWeekStolOneTwo.2
        OnValueChanged: execute { PLC_PRG_archive.x1 := TRUE; }
    Checkbox (653,106 113x35), "Среда", variable: NVI_RETAIN.dateWeekStolOneTwo.3
        OnValueChanged: execute { PLC_PRG_archive.x1 := TRUE; }
    Checkbox (653,141 113x35), "Четверг", variable: NVI_RETAIN.dateWeekStolOneTwo.4
        OnValueChanged: execute { PLC_PRG_archive.x1 := TRUE; }
    Checkbox (653,176 113x35), "Пятница", variable: NVI_RETAIN.dateWeekStolOneTwo.5
        OnValueChanged: execute { PLC_PRG_archive.x1 := TRUE; }
    Checkbox (653,211 113x35), "Суббота", variable: NVI_RETAIN.dateWeekStolOneTwo.6
        OnValueChanged: execute { PLC_PRG_archive.x1 := TRUE; }
    Checkbox (654,246 113x35), "Воскресенье", variable: NVI_RETAIN.dateWeekStolOneTwo.7
        OnValueChanged: execute { PLC_PRG_archive.x1 := TRUE; }
    Checkbox (653,2 238x35), "Активировать таймер", variable: NVI_RETAIN.dateWeekStolOneTwo.0
        OnValueChanged: execute { PLC_PRG_archive.x1 := TRUE; }
    Textfield (541,3 49x25), "Час"
    Textfield (598,3 49x25), "Мин"
    Textfield (541,38 49x30), "%d", text variable: NVI_RETAIN.hourMondayStolOne
        OnValueChanged: execute { PLC_PRG_archive.x1 := TRUE; }
        OnMouseClick: write the text variable via Default, min 0, max 23
    Textfield (598,38 49x30), "%d", text variable: NVI_RETAIN.minuteMondayStolOne
        OnValueChanged: execute { PLC_PRG_archive.x1 := TRUE; }
        OnMouseClick: write the text variable via Default, min 0, max 59
    Textfield (541,73 49x30), "%d", text variable: NVI_RETAIN.hourTuesdayStolOne
        OnValueChanged: execute { PLC_PRG_archive.x1 := TRUE; }
        OnMouseClick: write the text variable via Default, min 0, max 23
    Textfield (598,73 49x30), "%d", text variable: NVI_RETAIN.minuteTuesdayStolOne
        OnValueChanged: execute { PLC_PRG_archive.x1 := TRUE; }
        OnMouseClick: write the text variable via Default, min 0, max 59
    Textfield (541,108 49x30), "%d", text variable: NVI_RETAIN.hourWednesdayStolOne
        OnValueChanged: execute { PLC_PRG_archive.x1 := TRUE; }
        OnMouseClick: write the text variable via Default, min 0, max 23
    Textfield (541,143 49x30), "%d", text variable: NVI_RETAIN.hourThursdayStolOne
        OnValueChanged: execute { PLC_PRG_archive.x1 := TRUE; }
        OnMouseClick: write the text variable via Default, min 0, max 23
    Textfield (598,108 49x30), "%d", text variable: NVI_RETAIN.minuteWednesdayStolOne
        OnValueChanged: execute { PLC_PRG_archive.x1 := TRUE; }
        OnMouseClick: write the text variable via Default, min 0, max 59
    Textfield (541,213 49x30), "%d", text variable: NVI_RETAIN.hourSaturdayStolOne
        OnValueChanged: execute { PLC_PRG_archive.x1 := TRUE; }
        OnMouseClick: write the text variable via Default, min 0, max 23
    Textfield (598,178 49x30), "%d", text variable: NVI_RETAIN.minuteFridayStolOne
        OnValueChanged: execute { PLC_PRG_archive.x1 := TRUE; }
        OnMouseClick: write the text variable via Default, min 0, max 59
    Textfield (541,178 49x30), "%d", text variable: NVI_RETAIN.hourFridayStolOne
        OnValueChanged: execute { PLC_PRG_archive.x1 := TRUE; }
        OnMouseClick: write the text variable via Default, min 0, max 23
    Textfield (598,143 49x30), "%d", text variable: NVI_RETAIN.minuteThursdayStolOne
        OnValueChanged: execute { PLC_PRG_archive.x1 := TRUE; }
        OnMouseClick: write the text variable via Default, min 0, max 59
    Textfield (541,248 49x30), "%d", text variable: NVI_RETAIN.hourSundayStolOne
        OnValueChanged: execute { PLC_PRG_archive.x1 := TRUE; }
        OnMouseClick: write the text variable via Default, min 0, max 23
    Textfield (598,213 49x30), "%d", text variable: NVI_RETAIN.minuteSaturdayStolOne
        OnValueChanged: execute { PLC_PRG_archive.x1 := TRUE; }
        OnMouseClick: write the text variable via Default, min 0, max 59
    Textfield (598,248 49x30), "%d", text variable: NVI_RETAIN.minuteSundayStolOne
        OnValueChanged: execute { PLC_PRG_archive.x1 := TRUE; }
        OnMouseClick: write the text variable via Default, min 0, max 59
    PushSwitch (784,113 70x70), variable: PLC_PRG_Stol_1.START, behaviour: TAP, style: Switch-PushSwitch-Green
    Lamp1 (784,29 70x70), variable: PLC_PRG_Stol_1.INDIKATOR, style: Lamp-Lamp1-Blue
    PushSwitch (784,198 70x70), variable: PLC_PRG_Stol_1.STOP, behaviour: TAP, style: Switch-PushSwitch-Red
    Textfield (1314,316 0x1)
    Textfield (860,49 84x30), "РАБОТА"
    Textfield (860,133 94x30), "СТАРТ РУЧН."
    Textfield (860,218 84x30), "СТОП"
    DateRangeSelector (30,229 509x80)
        p758368661: dd.MM
        p2423372160: H:mm
        p1661464551: GenElemInst_30
    Textfield (648,431 76x30), "Pпод. %1.2f", text variable: PID_GLOBALS.g_rCurrentValue_Davlenie_Podacha_Stol_1_2
    Textfield (730,431 78x30), "Pобр. %1.2f", text variable: PID_GLOBALS.g_rCurrentValue_Davlenie_Obratnaja_Stol_1_2
        OnMouseClick: write the text variable via Default, min 0, max 100
    Textfield (817,431 73x30), "Δ Р %1.2f", text variable: PLC_PRG_CFC_Davlenie_Stol_1_2.Davlenie_Stol_1_2_rSetPoint
        OnValueChanged: execute { PLC_PRG_archive.x1 := TRUE; }
        OnMouseClick: write the text variable via Default, min 0, max 100
    Textfield (194,163 220x38), "Термостол №1"
    Textfield (648,361 108x30), "%d", text variable: PLC_PRG_Stol_1.Y2
        OnValueChanged: execute { PLC_PRG_archive.x1 := TRUE; }
        OnMouseClick: write the text variable via Default, min 0, max 100
    Image (898,-2 83x73), "HOME", image: VisuSymbols.Symbols.Home
        OnMouseClick:  Assign=HOME_1, Type=Assignment
    RoundedRectangle (895,429 48x34), "%1.2f", text variable: PLC_PRG_CFC_Davlenie_Stol_1_2.rCurrentValue
    RoundedRectangle (895,324 48x34), "%1.2f", text variable: PID_GLOBALS.g_rCurrentValue_Temperatura_Stol_1
    Lamp1 (950,315 24x23), variable: PLC_PRG_CFC_Temperatura_Stol_1.xMore, style: Lamp-Lamp1-Red
    Lamp1 (950,340 24x23), variable: PLC_PRG_CFC_Temperatura_Stol_1.xLess, style: Lamp-Lamp1-Blue
    Lamp1 (950,424 24x23), variable: PID_GLOBALS.xOut_More_Davlenie_Stol_1_2, style: Lamp-Lamp1-Blue
    Lamp1 (950,448 24x23), variable: PID_GLOBALS.xOut_Less_Davlenie_Stol_1_2, style: Lamp-Lamp1-Red
    Textfield (947,405 27x16), "ON"
    Textfield (947,298 27x16), "ON"
    Textfield (947,365 27x16), "OFF"
    Textfield (947,474 27x16), "OFF"
    Button (921,240 53x50), "?"
        OnMouseClick:  Assign=zapros, Type=Assignment
    Image (138,0 666x551), invisible if: Connection.warning = TRUE, image: VisuSymbols.Symbols.Caution
    Textfield (175,442 590x30), "МОДУЛЬ РАСШИРЕНИЯ В ОШИБКЕ!!!!!!!!!", invisible if: Connection.warning = TRUE
    Group (115,20 387x160), invisible if: PLC_PRG_archive.x1 = FALSE
        Rectangle (0,0 387x160), "Для того чтобы сохранить изменения нажмите да."
        Button (12,61 362x94), "ДА", invisible if: PLC_PRG_archive.x1 = FALSE
            tap PID_GLOBALS.zGO
            OnMouseClick: execute { PLC_PRG_archive.x1 := FALSE; }
END_VISUALIZATION

// Device/Application/Parostol_Zadanie/HOME_1
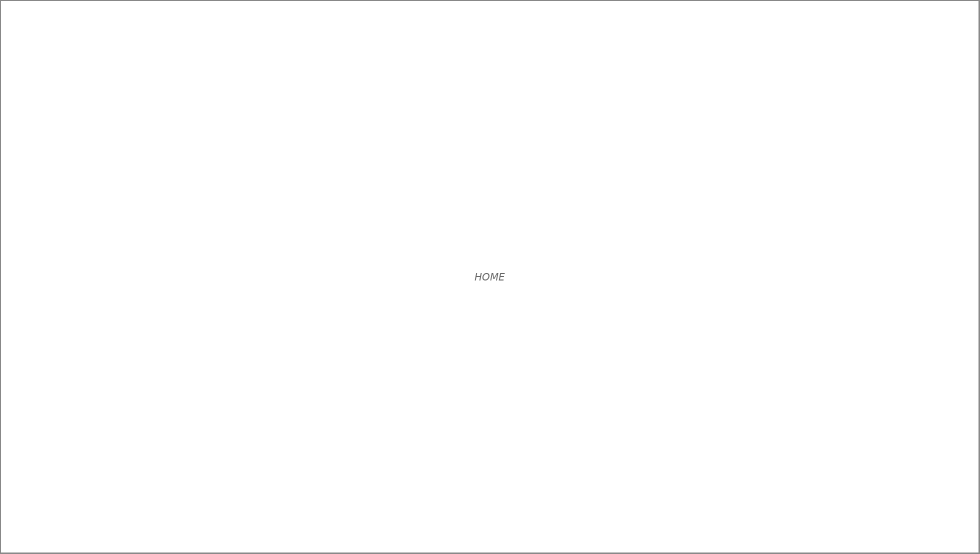
VISUALIZATION HOME_1  // 980x554
VAR_IN_OUT
END_VAR
VAR
	bResetTrigger : BOOL;
	bStart : BOOL;
	bStop : BOOL;
	bStore : BOOL;
	sStoreFilename : STRING;
	bRestore : BOOL;
	sRestoreFilename : STRING;
END_VAR
    TabControl (0,0 980x554)
        shows HOME()
        shows MnemoScheme()
        shows Journal()
        shows Visualization_CFC_Temperatura()
        shows Visualization_CFC_Davlenie()
        [0]: TabTitle=Главная
        [1]: TabTitle=Мнемосхема
        [2]: TabTitle=Журнал тревог
        [3]: TabTitle=ПИД t Стол 1
        [4]: TabTitle=Пид P Стол 1
    Textfield (1314,316 0x1)
END_VISUALIZATION

// Device/Application/Parostol_Zadanie/Visualization_CFC_Davlenie_1_2
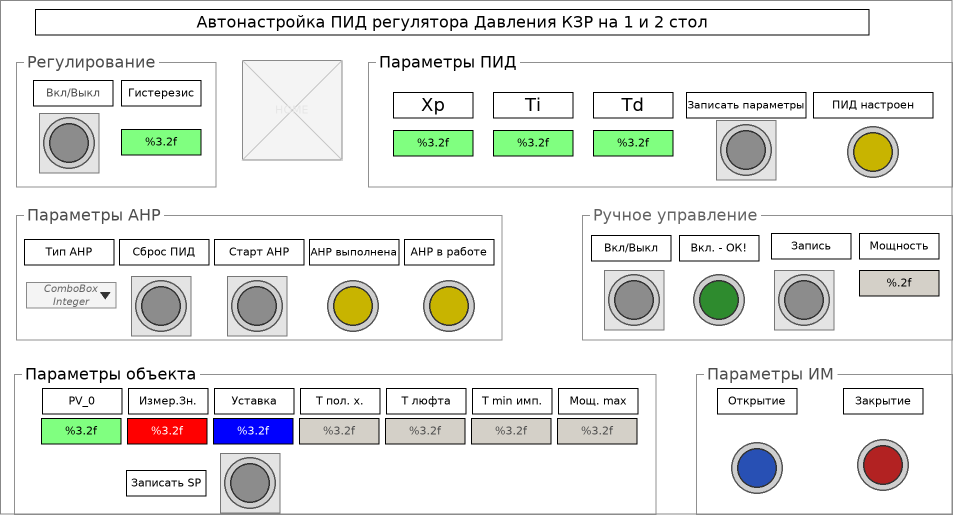
VISUALIZATION Visualization_CFC_Davlenie_1_2  // 953x515
    GroupBox (16,207 486x133), "Параметры АНР"
        Rectangle (293,32 90x26), "АНР выполнена"
        Lamp1 (307,69 60x60), variable: PLC_PRG_CFC_Davlenie_Stol_1_2.xAutotuneCompleted, style: Lamp-Lamp1-Yellow
        Rectangle (103,32 90x26), "Сброс ПИД"
        PushSwitchLed (211,69 60x60), variable: PLC_PRG_CFC_Davlenie_Stol_1_2.xStartAutotune, behaviour: TOGGLE, style: Switch-PushSwitchLed-Gray
        PushSwitch (115,69 60x60), variable: PLC_PRG_CFC_Davlenie_Stol_1_2.xReset, behaviour: TAP, style: Switch-PushSwitch-Gray
        Rectangle (388,32 90x26), "АНР в работе"
        Lamp1 (403,69 60x60), variable: PLC_PRG_CFC_Davlenie_Stol_1_2.xAutotuneInProgress, style: Lamp-Lamp1-Yellow
        Rectangle (198,32 90x26), "Старт АНР"
        ComboBoxInteger (10,75 90x26), variable: PLC_PRG_CFC_Davlenie_Stol_1_2.eAutotuneMode, text list: 'ANR_MODE'
    Rectangle (24,239 90x26), "Тип АНР"
    GroupBox (16,54 200x133), "Регулирование"
        PushSwitchLed (23,59 60x60), variable: PLC_PRG_CFC_Davlenie_Stol_1_2.xIsEnabledPid, behaviour: TOGGLE, style: Switch-PushSwitchLed-Gray
        Rectangle (105,26 80x26), "Гистерезис"
        RoundedRectangle (105,75 80x26), "%3.2f", text variable: PLC_PRG_CFC_Davlenie_Stol_1_2.rDeadBand
            OnMouseClick: write the text variable via Default
    Rectangle (33,80 80x26), "Вкл/Выкл"
    GroupBox (368,54 585x133), "Параметры ПИД"
        Lamp1 (475,68 60x60), variable: PLC_PRG_CFC_Davlenie_Stol_1_2.xIsPidValidSettings, style: Lamp-Lamp1-Yellow
        PushSwitch (348,66 60x60), variable: PLC_PRG_CFC_Davlenie_Stol_1_2.xWritePidSettings, behaviour: TAP, style: Switch-PushSwitch-Gray
        Rectangle (318,38 120x26), "Записать параметры"
        Rectangle (445,38 120x26), "ПИД настроен"
    RoundedRectangle (393,130 80x26), "%3.2f", text variable: PLC_PRG_CFC_Davlenie_Stol_1_2.rXp
        OnMouseClick: write the text variable via Default
    RoundedRectangle (493,130 80x26), "%3.2f", text variable: PLC_PRG_CFC_Davlenie_Stol_1_2.rTi
        OnMouseClick: write the text variable via Default
    RoundedRectangle (593,130 80x26), "%3.2f", text variable: PLC_PRG_CFC_Davlenie_Stol_1_2.rTd
        OnMouseClick: write the text variable via Default
    Rectangle (393,92 80x26), "Xp"
    Rectangle (493,92 80x26), "Ti"
    Rectangle (593,92 80x26), "Td"
    GroupBox (696,366 257x149), "Параметры ИМ"
        Rectangle (21,22 80x26), "Открытие"
        Rectangle (147,22 80x26), "Закрытие"
        Lamp1 (31,72 60x60), variable: PID_GLOBALS.xOut_More_Davlenie_Stol_1_2, style: Lamp-Lamp1-Blue
        Lamp1 (157,69 60x60), variable: PID_GLOBALS.xOut_Less_Davlenie_Stol_1_2, style: Lamp-Lamp1-Red
    GroupBox (14,366 642x149), "Параметры объекта"
        RoundedRectangle (113,52 80x26), "%3.2f", text variable: PLC_PRG_CFC_Davlenie_Stol_1_2.rCurrentValue
        RoundedRectangle (371,52 80x26), "%3.2f", text variable: PLC_PRG_CFC_Davlenie_Stol_1_2.rTluft
            OnMouseClick: write the text variable via Default
        RoundedRectangle (543,52 80x26), "%3.2f", text variable: PLC_PRG_CFC_Davlenie_Stol_1_2.rDy_anr
            OnMouseClick: write the text variable via Default
        PushSwitch (206,87 60x60), variable: PLC_PRG_CFC_Davlenie_Stol_1_2.xSetSP, behaviour: TAP, style: Switch-PushSwitch-Gray
        Rectangle (112,104 80x26), "Записать SP"
        Rectangle (200,22 80x26), "Уставка", tooltip "Уставка давления"
        RoundedRectangle (199,52 80x26), "%3.2f", text variable: PLC_PRG_CFC_Davlenie_Stol_1_2.Davlenie_Stol_1_2_rSetPoint
            OnMouseClick: write the text variable via Default
        RoundedRectangle (457,52 80x26), "%3.2f", text variable: PLC_PRG_CFC_Davlenie_Stol_1_2.rTimp
            OnMouseClick: write the text variable via Default
        RoundedRectangle (285,52 80x26), "%3.2f", text variable: PLC_PRG_CFC_Davlenie_Stol_1_2.rTval
            OnMouseClick: write the text variable via Default
    RoundedRectangle (41,418 80x26), "%3.2f", text variable: PLC_PRG_CFC_Davlenie_Stol_1_2.rSteadyValue
        OnMouseClick: write the text variable via Default
    Rectangle (42,388 80x26), "PV_0", tooltip "Значение регулируемого параметра при нулевом уровне мощности (при Y=0)"
    Rectangle (128,388 80x26), "Измер.Зн.", tooltip "Значение давления"
    Rectangle (300,388 80x26), "Т пол. х.", tooltip "Время полного хода ИМ, сек."
    Rectangle (386,388 80x26), "Т люфта", tooltip "Время выборки люфта ИМ, сек."
    Rectangle (472,388 80x26), "Т min имп.", tooltip "Минимальная длительность импульса, сек."
    Rectangle (558,388 80x26), "Мощ. max", tooltip "Размах мощности (в процентах), выдаваемый на задвижку от текущей позиции при АНР. Например, при положении задвижки 50% и значении DY_ANR=25% в ходе АНР задвижка будет перемещаться от 25 до 75% (без учета влияния физических процессов на перемещение задвижки) Диапазон возможныз значений: 0.0...100.0 (%)"
    GroupBox (582,207 371x133), "Ручное управление"
        PushSwitchLed (22,63 60x60), variable: PLC_PRG_CFC_Davlenie_Stol_1_2.xManualMode, behaviour: TOGGLE, style: Switch-PushSwitchLed-Gray
        PushSwitch (192,63 60x60), variable: PLC_PRG_CFC_Davlenie_Stol_1_2.xManual_set, behaviour: TAP, style: Switch-PushSwitch-Gray
        Rectangle (189,26 80x26), "Запись"
        RoundedRectangle (277,63 80x26), "%.2f", text variable: PLC_PRG_CFC_Davlenie_Stol_1_2.rManual_mean
            OnMouseClick: write the text variable via Default
        Rectangle (277,26 80x26), "Мощность"
        Lamp1 (107,63 60x60), variable: PLC_PRG_CFC_Davlenie_Stol_1_2.xSetManualOK, style: Lamp-Lamp1-Green
        Rectangle (9,28 80x26), "Вкл/Выкл"
        Rectangle (97,28 80x26), "Вкл. - ОК!"
    Rectangle (35,9 834x26), "Автонастройка ПИД регулятора Давления КЗР на 1 и 2 стол"
    Image (242,60 100x100), "HOME", image: VisuSymbols.Symbols.Home
        OnMouseClick:  Assign=HOME_1, Type=Assignment
END_VISUALIZATION

// Device/Application/Parostol_Zadanie/HOME
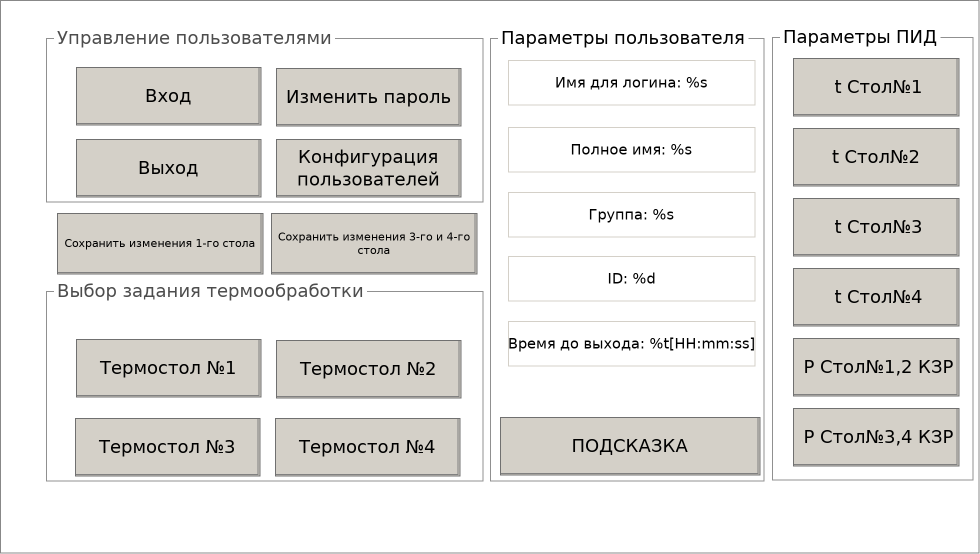
VISUALIZATION HOME  // 980x554
    GroupBox (772,29 201x451), "Параметры ПИД"
        Button (21,379 166x58), "Р Стол№3,4 КЗР"
            OnMouseClick:  Assign=Visualization_CFC_Davlenie_3_4, Type=Assignment
        Button (21,29 166x58), "t Стол№1"
            OnMouseClick:  Assign=Visualization_CFC_Temperatura_1, Type=Assignment
    GroupBox (46,30 437x172), "Управление пользователями"
        Button (230,109 185x58), "Конфигурация пользователей"
            OnMouseClick:  Type=OpenUserConfiguration
    GroupBox (46,283 437x198), "Выбор задания термообработки"
        Button (30,56 185x58), "Термостол №1"
            OnMouseClick:  Assign=Zadanie_1, Type=Assignment
        Button (230,57 185x58), "Термостол №2"
            OnMouseClick:  Assign=Zadanie_2, Type=Assignment
        Button (29,135 185x58), "Термостол №3"
            OnMouseClick:  Assign=Zadanie_3, Type=Assignment
        Button (229,135 185x58), "Термостол №4"
            OnMouseClick:  Assign=Zadanie_4, Type=Assignment
    Button (76,67 185x58), "Вход"
        OnMouseClick:  Type=Login
    Button (76,139 185x58), "Выход"
        OnMouseClick:  Type=Logout
    Button (276,68 185x58), "Изменить пароль"
        OnMouseClick:  Type=ChangeUserPassword
    GroupBox (490,30 274x451), "Параметры пользователя"
        Textfield (18,291 247x45), "Время до выхода: %t[HH:mm:ss]", text variable: VisuElems.CurrentRemainingAutoLogoutTime, invisible if: NOT(VisuElems.CurrentUseAutoLogoutTime)
        Textfield (18,97 247x45), "Полное имя: %s", text variable: VisuElems.CurrentFullUserName
        Textfield (18,162 247x45), "Группа: %s", text variable: VisuElems.CurrentUserGroupName
        Textfield (18,226 247x45), "ID: %d", text variable: VisuElems.CurrentUserGroupId
        Button (10,387 260x58), "ПОДСКАЗКА"
            OnMouseClick:  Assign=instrykcai_avtoriz, Type=Assignment
    Textfield (508,60 247x45), "Имя для логина: %s", text variable: VisuElems.CurrentUserName
    Button (793,128 166x58), "t Стол№2"
    Button (793,198 166x58), "t Стол№3"
        OnMouseClick:  Assign=Visualization_CFC_Temperatura_3, Type=Assignment
    Button (793,268 166x58), "t Стол№4"
        OnMouseClick:  Assign=Visualization_CFC_Temperatura_4, Type=Assignment
    Button (793,338 166x58), "Р Стол№1,2 КЗР"
        OnMouseClick:  Assign=Visualization_CFC_Davlenie_1_2, Type=Assignment
    Button (271,213 206x61), "Сохранить изменения 3-го и 4-го стола"
        tap PID_GLOBALS.yGO
        OnMouseClick: execute { PLC_PRG_archive.z1 := FALSE; PLC_PRG_archive.y1 := FALSE; }
    Button (57,213 206x61), "Сохранить изменения 1-го стола"
        tap PID_GLOBALS.zGO
        OnMouseClick: execute { PLC_PRG_archive.x1 := FALSE; }
END_VISUALIZATION

// Device/Application/Parostol_Zadanie/MnemoScheme
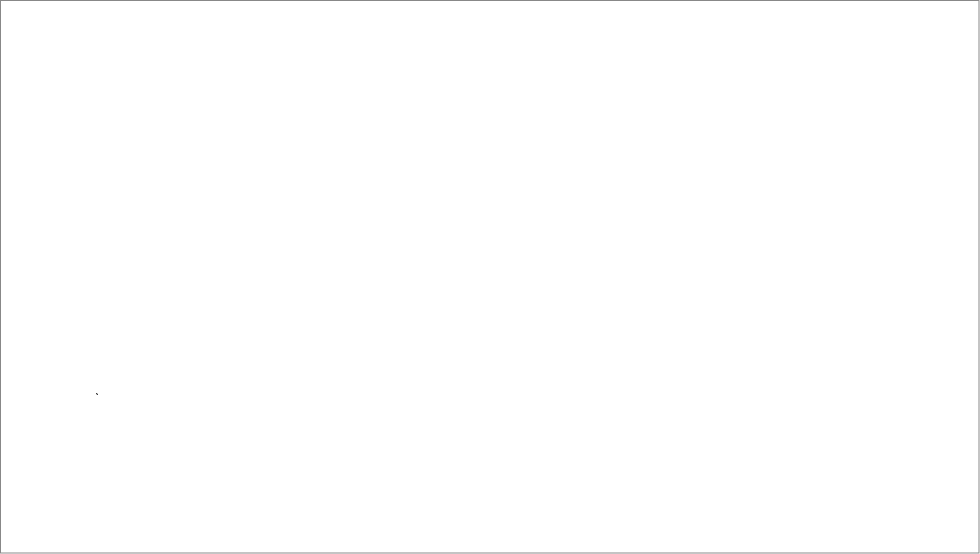
VISUALIZATION MnemoScheme  // 980x554
    Polygon (96,393) (97,394)
END_VISUALIZATION

// Device/Application/Parostol_Zadanie/Journal
VISUALIZATION Journal  // 980x554
END_VISUALIZATION

// Device/Application/Parostol_Zadanie/Zadanie_2
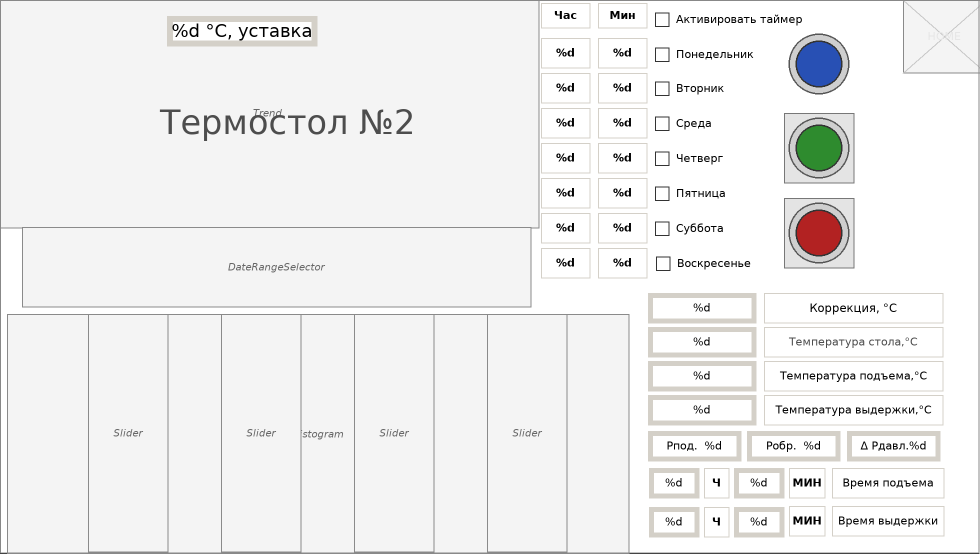
VISUALIZATION Zadanie_2  // 980x554
VAR_IN_OUT
END_VAR
VAR
	bResetTrigger : BOOL;
	bStart : BOOL;
	bStop : BOOL;
	bStore : BOOL;
	sStoreFilename : STRING;
	bRestore : BOOL;
	sRestoreFilename : STRING;
END_VAR
    Rectangle (-1,0 980x554)
    Histogram (7,314 622x240), scale format: %.1f, scale 0..100
        p518627256: °C
        p1518820177: PLC_PRG_Stol_2.arrHist1
        p102497268: PLC_PRG_1.arrHist1
        p788070771: ARRAY [0..3] OF REAL
    Slider (88,314 80x238), variable: PLC_PRG_Stol_2.Y1, scale 0..100
    Slider (221,314 80x238), variable: PLC_PRG_Stol_2.Y2, scale 0..100
    Slider (354,314 80x238), variable: PLC_PRG_Stol_2.Y3, scale 0..100
    Slider (487,314 80x238), variable: PLC_PRG_Stol_2.Y4, scale 0..100
    Trend (-4,-2 543x230)
        p758368661: dd.MM.yyyy
        p2423372160: H:mm:ss
        p2833066001: Visualization_Trend_Stol_2
        p2059293862: GenElemInst_240
    Line (925,485)
    Textfield (648,293 108x30), "%d"
        OnMouseClick: write the text variable via Default
    Textfield (648,395 108x30), "%d", text variable: PLC_PRG_Stol_2.Y3
        OnMouseClick: write the text variable via Default, min 0, max 100
    Textfield (648,327 108x30), "%d", text variable: PLC_PRG_Stol_2.Y1
        OnMouseClick: write the text variable via Default, min 0, max 100
    Textfield (649,468 50x30), "%d", text variable: PLC_PRG_Stol_2.HX2
        OnMouseClick: write the text variable via Default, min 0
    Textfield (764,293 179x30), "Коррекция, °C"
    Textfield (764,327 179x30), "Температура стола,°C"
    Textfield (764,361 179x30), "Температура подъема,°C"
    Textfield (764,395 179x30), "Температура выдержки,°C"
    Textfield (832,468 112x30), "Время подъема"
    Textfield (649,507 50x30), "%d", text variable: PLC_PRG_Stol_2.HX3
        OnMouseClick: write the text variable via Default, min 0
    Textfield (832,506 112x30), "Время выдержки"
    Textfield (167,16 150x30), "%d °C, уставка", text variable: PID_GLOBALS.Temperatura_Stol_2_rSetPoint
    Textfield (734,468 50x30), "%d", text variable: PLC_PRG_Stol_2.MX2
        OnMouseClick: write the text variable via Default, min 0, max 59
    Textfield (704,468 25x30), "Ч"
    Textfield (789,468 36x30), "МИН"
    Textfield (734,507 50x30), "%d", text variable: PLC_PRG_Stol_2.MX3
        OnMouseClick: write the text variable via Default, min 0, max 59
    Textfield (704,507 25x30), "Ч"
    Textfield (789,506 36x30), "МИН"
    Checkbox (653,37 113x35), "Понедельник", variable: PLC_PRG_Stol_2.PONEDEL
    Checkbox (653,71 113x35), "Вторник", variable: PLC_PRG_Stol_2.VTORN
    Checkbox (653,106 113x35), "Среда", variable: PLC_PRG_Stol_2.SREDA
    Checkbox (653,141 113x35), "Четверг", variable: PLC_PRG_Stol_2.CHETV
    Checkbox (653,176 113x35), "Пятница", variable: PLC_PRG_Stol_2.PJATN
    Checkbox (653,211 113x35), "Суббота", variable: PLC_PRG_Stol_2.SUBB
    Checkbox (654,246 113x35), "Воскресенье", variable: PLC_PRG_Stol_2.VOSKR
    Checkbox (653,2 233x35), "Активировать таймер", variable: PLC_PRG_Stol_2.ACTIVATOR_TIMER
    Textfield (541,3 49x25), "Час"
    Textfield (598,3 49x25), "Мин"
    Textfield (541,38 49x30), "%d", text variable: PLC_PRG_Stol_2.HOUR_PONEDEL
        OnMouseClick: write the text variable via Default, min 0, max 23
    Textfield (598,38 49x30), "%d", text variable: PLC_PRG_Stol_2.MINUTE_PONEDEL
        OnMouseClick: write the text variable via Default, min 0, max 59
    Textfield (541,73 49x30), "%d", text variable: PLC_PRG_Stol_2.HOUR_VTORN
        OnMouseClick: write the text variable via Default, min 0, max 23
    Textfield (598,73 49x30), "%d", text variable: PLC_PRG_Stol_2.MINUTE_VTORN
        OnMouseClick: write the text variable via Default, min 0, max 59
    Textfield (541,108 49x30), "%d", text variable: PLC_PRG_Stol_2.HOUR_SREDA
        OnMouseClick: write the text variable via Default, min 0, max 23
    Textfield (541,143 49x30), "%d", text variable: PLC_PRG_Stol_2.HOUR_CHETV
        OnMouseClick: write the text variable via Default, min 0, max 23
    Textfield (598,108 49x30), "%d", text variable: PLC_PRG_Stol_2.MINUTE_SREDA
        OnMouseClick: write the text variable via Default, min 0, max 59
    Textfield (541,213 49x30), "%d", text variable: PLC_PRG_Stol_2.HOUR_SUBB
        OnMouseClick: write the text variable via Default, min 0, max 23
    Textfield (598,178 49x30), "%d", text variable: PLC_PRG_Stol_2.MINUTE_PJATN
        OnMouseClick: write the text variable via Default, min 0, max 59
    Textfield (541,178 49x30), "%d", text variable: PLC_PRG_Stol_2.HOUR_PJATN
        OnMouseClick: write the text variable via Default, min 0, max 23
    Textfield (598,143 49x30), "%d", text variable: PLC_PRG_Stol_2.MINUTE_CHETV
        OnMouseClick: write the text variable via Default, min 0, max 59
    Textfield (541,248 49x30), "%d", text variable: PLC_PRG_Stol_2.HOUR_VOSKR
        OnMouseClick: write the text variable via Default, min 0, max 23
    Textfield (598,213 49x30), "%d", text variable: PLC_PRG_Stol_2.MINUTE_SUBB
        OnMouseClick: write the text variable via Default, min 0, max 59
    Textfield (598,248 49x30), "%d", text variable: PLC_PRG_Stol_2.MINUTE_VOSKR
        OnMouseClick: write the text variable via Default, min 0, max 59
    PushSwitch (784,113 70x70), variable: PLC_PRG_Stol_2.START, behaviour: TAP, style: Switch-PushSwitch-Green
    Lamp1 (784,29 70x70), variable: PLC_PRG_Stol_2.INDIKATOR, style: Lamp-Lamp1-Blue
    PushSwitch (784,198 70x70), variable: PLC_PRG_Stol_2.STOP, behaviour: TAP, style: Switch-PushSwitch-Red
    Textfield (1314,316 0x1)
    Textfield (860,49 84x30), "РАБОТА"
    Textfield (860,133 94x30), "СТАРТ РУЧН."
    Textfield (860,218 84x30), "СТОП"
    DateRangeSelector (22,227 509x80)
        p758368661: dd.MM
        p2423372160: H:mm
        p1661464551: GenElemInst_30
    Textfield (648,431 93x30), "Pпод. %d", text variable: PID_GLOBALS.g_rCurrentValue_Davlenie_Podacha_Stol_1_2
        OnMouseClick: write the text variable via Default, min 0, max 100
    Textfield (747,431 93x30), "Pобр. %d", text variable: PID_GLOBALS.g_rCurrentValue_Davlenie_Obratnaja_Stol_1_2
        OnMouseClick: write the text variable via Default, min 0, max 100
    Textfield (847,431 93x30), "Δ Рдавл.%d", text variable: PID_GLOBALS.Davlenie_Stol_1_2_rSetPoint
        OnMouseClick: write the text variable via Default, min 0, max 100
    Textfield (149,103 278x38), "Термостол №2"
    Textfield (648,361 108x30), "%d", text variable: PLC_PRG_Stol_2.Y2
        OnMouseClick: write the text variable via Default, min 0, max 100
    Image (903,0 83x73), "HOME", image: VisuSymbols.Symbols.Home
        OnMouseClick:  Assign=HOME_1, Type=Assignment
END_VISUALIZATION

// Device/Application/Parostol_Zadanie/Visualization_CFC_Temperatura_1
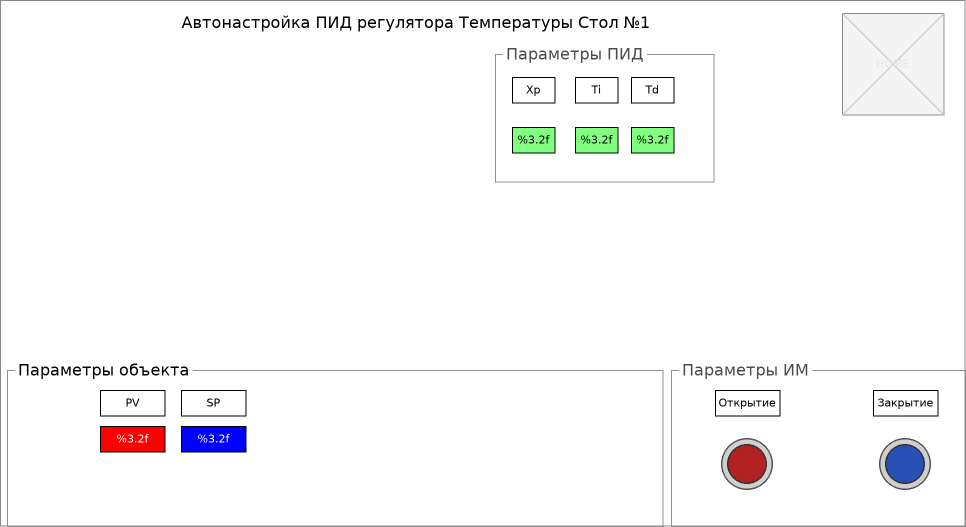
VISUALIZATION Visualization_CFC_Temperatura_1  // 966x527
    GroupBox (7,362 656x165), "Параметры объекта"
        RoundedRectangle (93,64 65x26), "%3.2f", text variable: PID_GLOBALS.g_rCurrentValue_Temperatura_Stol_1
    GroupBox (495,46 219x136), "Параметры ПИД"
        RoundedRectangle (136,81 43x26), "%3.2f", text variable: PLC_PRG_CFC_Temperatura_Stol_1.rTd
            OnMouseClick: write the text variable via Default
        RoundedRectangle (80,81 43x26), "%3.2f", text variable: PLC_PRG_CFC_Temperatura_Stol_1.rTi
            OnMouseClick: write the text variable via Default
        RoundedRectangle (17,81 43x26), "%3.2f", text variable: PLC_PRG_CFC_Temperatura_Stol_1.rXp
            OnMouseClick: write the text variable via Default
        Rectangle (17,31 43x26), "Xp"
        Rectangle (80,31 43x26), "Ti"
        Rectangle (136,31 43x26), "Td"
    RoundedRectangle (181,426 65x26), "%3.2f", text variable: PLC_PRG_Stol_1.Y1
        OnMouseClick: write the text variable via Default
    Rectangle (100,390 65x26), "PV", tooltip "Значение температуры"
    Rectangle (181,390 65x26), "SP", tooltip "Уставка температуры"
    GroupBox (671,362 295x165), "Параметры ИМ"
        Rectangle (44,28 65x26), "Открытие"
        Rectangle (202,28 65x26), "Закрытие"
        Lamp1 (46,72 60x60), variable: PLC_PRG_CFC_Temperatura_Stol_1.xMore, style: Lamp-Lamp1-Red
        Lamp1 (204,72 60x60), variable: PLC_PRG_CFC_Temperatura_Stol_1.xLess, style: Lamp-Lamp1-Blue
    Image (842,13 102x102), "HOME", image: VisuSymbols.Symbols.Home
        OnMouseClick:  Assign=HOME_1, Type=Assignment
    Rectangle (107,7 618x31), "Автонастройка ПИД регулятора Температуры Стол №1"
END_VISUALIZATION

// Device/Application/Parostol_Zadanie/Zadanie_3
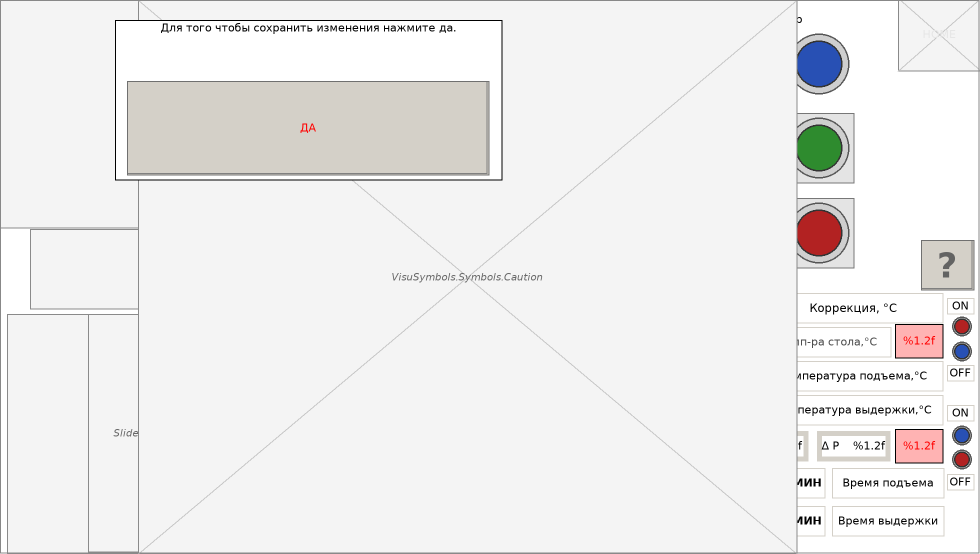
VISUALIZATION Zadanie_3  // 980x554
VAR_IN_OUT
END_VAR
VAR
	bResetTrigger : BOOL;
	bStart : BOOL;
	bStop : BOOL;
	bStore : BOOL;
	sStoreFilename : STRING;
	bRestore : BOOL;
	sRestoreFilename : STRING;
END_VAR
    Rectangle (0,-1 980x554)
    Histogram (7,314 622x240), scale format: %.1f, scale 0..100
        p518627256: °C
        p1518820177: PLC_PRG_Stol_3.arrHist1
        p102497268: PLC_PRG_Stol_3.arrHist1
        p788070771: ARRAY [0..3] OF REAL
    Slider (88,314 80x238), variable: PLC_PRG_Stol_3.Y1, scale 0..100
        OnValueChanged: execute { PLC_PRG_archive.y1 := TRUE; }
    Slider (215,313 80x238), variable: PLC_PRG_Stol_3.Y2, scale 0..100
        OnValueChanged: execute { PLC_PRG_archive.y1 := TRUE; }
    Slider (354,314 80x238), variable: PLC_PRG_Stol_3.Y3, scale 0..100
        OnValueChanged: execute { PLC_PRG_archive.y1 := TRUE; }
    Slider (487,314 80x238), variable: PLC_PRG_Stol_3.Y4, scale 0..100
        OnValueChanged: execute { PLC_PRG_archive.y1 := TRUE; }
    Trend (-3,-2 543x230)
        p758368661: dd.MM.yyyy
        p2423372160: H:mm:ss
        p2833066001: Visualization_Trend_Stol_3
        p2059293862: GenElemInst_240
    Line (925,485)
    Textfield (648,293 108x30)
        OnMouseClick: write the text variable via Default
    Textfield (648,395 108x30), "%d", text variable: PLC_PRG_Stol_3.Y3
        OnValueChanged: execute { PLC_PRG_archive.y1 := TRUE; }
        OnMouseClick: write the text variable via Default, min 0, max 100
    Textfield (648,327 108x30), "%d", text variable: PLC_PRG_Stol_3.Y1
        OnValueChanged: execute { PLC_PRG_archive.y1 := TRUE; }
        OnMouseClick: write the text variable via Default, min 0, max 100
    Textfield (649,468 50x30), "%d", text variable: PLC_PRG_Stol_3.HX2
        OnValueChanged: execute { PLC_PRG_archive.y1 := TRUE; }
        OnMouseClick: write the text variable via Default, min 0
    Textfield (764,293 179x30), "Коррекция, °C"
    Textfield (764,327 127x30), "Темп-ра стола,°C"
    Textfield (764,361 179x30), "Температура подъема,°C"
    Textfield (764,395 179x30), "Температура выдержки,°C"
    Textfield (832,468 112x30), "Время подъема"
    Textfield (649,507 50x30), "%d", text variable: PLC_PRG_Stol_3.HX3
        OnValueChanged: execute { PLC_PRG_archive.y1 := TRUE; }
        OnMouseClick: write the text variable via Default, min 0
    Textfield (832,506 112x30), "Время выдержки"
    Textfield (167,16 150x30), "%d °C, уставка", text variable: PID_GLOBALS.Temperatura_Stol_3_rSetPoint
    Textfield (734,468 50x30), "%d", text variable: PLC_PRG_Stol_3.MX2
        OnValueChanged: execute { PLC_PRG_archive.y1 := TRUE; }
        OnMouseClick: write the text variable via Default, min 0, max 59
    Textfield (704,468 25x30), "Ч"
    Textfield (789,468 36x30), "МИН"
    Textfield (734,507 50x30), "%d", text variable: PLC_PRG_Stol_3.MX3
        OnValueChanged: execute { PLC_PRG_archive.y1 := TRUE; }
        OnMouseClick: write the text variable via Default, min 0, max 59
    Textfield (704,507 25x30), "Ч"
    Textfield (789,506 36x30), "МИН"
    Checkbox (653,37 113x35), "Понедельник", variable: NVI_RETAIN.dateWeekStolThreeFour.1
        OnValueChanged: execute { PLC_PRG_archive.y1 := TRUE; }
    Checkbox (653,71 113x35), "Вторник", variable: NVI_RETAIN.dateWeekStolThreeFour.2
        OnValueChanged: execute { PLC_PRG_archive.y1 := TRUE; }
    Checkbox (653,106 113x35), "Среда", variable: NVI_RETAIN.dateWeekStolThreeFour.3
        OnValueChanged: execute { PLC_PRG_archive.y1 := TRUE; }
    Checkbox (653,141 113x35), "Четверг", variable: NVI_RETAIN.dateWeekStolThreeFour.4
        OnValueChanged: execute { PLC_PRG_archive.y1 := TRUE; }
    Checkbox (653,176 113x35), "Пятница", variable: NVI_RETAIN.dateWeekStolThreeFour.5
        OnValueChanged: execute { PLC_PRG_archive.y1 := TRUE; }
    Checkbox (653,211 113x35), "Суббота", variable: NVI_RETAIN.dateWeekStolThreeFour.6
        OnValueChanged: execute { PLC_PRG_archive.y1 := TRUE; }
    Checkbox (653,246 113x35), "Воскресенье", variable: NVI_RETAIN.dateWeekStolThreeFour.7
        OnValueChanged: execute { PLC_PRG_archive.y1 := TRUE; }
    Checkbox (653,2 234x35), "Активировать таймер", variable: NVI_RETAIN.dateWeekStolThreeFour.0
        OnValueChanged: execute { PLC_PRG_archive.y1 := TRUE; }
    Textfield (541,3 49x25), "Час"
    Textfield (598,3 49x25), "Мин"
    Textfield (541,38 49x30), "%d", text variable: NVI_RETAIN.hourMondayStolThree
        OnValueChanged: execute { PLC_PRG_archive.y1 := TRUE; }
        OnMouseClick: write the text variable via Default, min 0, max 23
    Textfield (598,38 49x30), "%d", text variable: NVI_RETAIN.minuteMondayStolThree
        OnValueChanged: execute { PLC_PRG_archive.y1 := TRUE; }
        OnMouseClick: write the text variable via Default, min 0, max 59
    Textfield (541,73 49x30), "%d", text variable: NVI_RETAIN.hourTuesdayStolThree
        OnValueChanged: execute { PLC_PRG_archive.y1 := TRUE; }
        OnMouseClick: write the text variable via Default, min 0, max 23
    Textfield (598,73 49x30), "%d", text variable: NVI_RETAIN.minuteTuesdayStolThree
        OnValueChanged: execute { PLC_PRG_archive.y1 := TRUE; }
        OnMouseClick: write the text variable via Default, min 0, max 59
    Textfield (541,108 49x30), "%d", text variable: NVI_RETAIN.hourWednesdayStolThree
        OnValueChanged: execute { PLC_PRG_archive.y1 := TRUE; }
        OnMouseClick: write the text variable via Default, min 0, max 23
    Textfield (541,143 49x30), "%d", text variable: NVI_RETAIN.hourThursdayStolThree
        OnValueChanged: execute { PLC_PRG_archive.y1 := TRUE; }
        OnMouseClick: write the text variable via Default, min 0, max 23
    Textfield (598,108 49x30), "%d", text variable: NVI_RETAIN.minuteWednesdayStolThree
        OnValueChanged: execute { PLC_PRG_archive.y1 := TRUE; }
        OnMouseClick: write the text variable via Default, min 0, max 59
    Textfield (541,213 49x30), "%d", text variable: NVI_RETAIN.hourSaturdayStolThree
        OnValueChanged: execute { PLC_PRG_archive.y1 := TRUE; }
        OnMouseClick: write the text variable via Default, min 0, max 23
    Textfield (598,178 49x30), "%d", text variable: NVI_RETAIN.minuteFridayStolThree
        OnValueChanged: execute { PLC_PRG_archive.y1 := TRUE; }
        OnMouseClick: write the text variable via Default, min 0, max 59
    Textfield (541,178 49x30), "%d", text variable: NVI_RETAIN.hourFridayStolThree
        OnValueChanged: execute { PLC_PRG_archive.y1 := TRUE; }
        OnMouseClick: write the text variable via Default, min 0, max 23
    Textfield (598,143 49x30), "%d", text variable: NVI_RETAIN.minuteThursdayStolThree
        OnValueChanged: execute { PLC_PRG_archive.y1 := TRUE; }
        OnMouseClick: write the text variable via Default, min 0, max 59
    Textfield (541,248 49x30), "%d", text variable: NVI_RETAIN.hourSundayStolThree
        OnValueChanged: execute { PLC_PRG_archive.y1 := TRUE; }
        OnMouseClick: write the text variable via Default, min 0, max 23
    Textfield (598,213 49x30), "%d", text variable: NVI_RETAIN.minuteSaturdayStolThree
        OnValueChanged: execute { PLC_PRG_archive.y1 := TRUE; }
        OnMouseClick: write the text variable via Default, min 0, max 59
    Textfield (598,248 49x30), "%d", text variable: NVI_RETAIN.minuteSundayStolThree
        OnValueChanged: execute { PLC_PRG_archive.y1 := TRUE; }
        OnMouseClick: write the text variable via Default, min 0, max 59
    PushSwitch (784,113 70x70), variable: PLC_PRG_Stol_3.START, behaviour: TAP, style: Switch-PushSwitch-Green
    Lamp1 (784,29 70x70), variable: PLC_PRG_Stol_3.INDIKATOR, style: Lamp-Lamp1-Blue
    PushSwitch (784,198 70x70), variable: PLC_PRG_Stol_3.STOP, behaviour: TAP, style: Switch-PushSwitch-Red
    Textfield (1314,316 0x1)
    Textfield (860,49 84x30), "РАБОТА"
    Textfield (860,133 94x30), "СТАРТ РУЧН."
    Textfield (860,218 84x30), "СТОП"
    DateRangeSelector (30,229 509x80)
        p758368661: dd.MM
        p2423372160: H:mm
        p1661464551: GenElemInst_30
    Textfield (648,431 76x30), "Pобр. %1.2f", text variable: PID_GLOBALS.g_rCurrentValue_Davlenie_Podacha_Stol_3_4
    Textfield (730,431 78x30), "Pпод. %1.2f", text variable: PID_GLOBALS.g_rCurrentValue_Davlenie_Obratnaja_Stol_3_4
        OnMouseClick: write the text variable via Default, min 0, max 100
    Textfield (817,431 73x30), "Δ Р %1.2f", text variable: PLC_PRG_CFC_Davlenie_Stol_3_4.Davlenie_Stol_3_4_rSetPoint
        OnValueChanged: execute { PLC_PRG_archive.y1 := TRUE; }
        OnMouseClick: write the text variable via Default, min 0, max 100
    Textfield (168,163 220x38), "Термостол №3"
    Textfield (648,361 108x30), "%d", text variable: PLC_PRG_Stol_3.Y2
        OnValueChanged: execute { PLC_PRG_archive.y1 := TRUE; }
        OnMouseClick: write the text variable via Default, min 0, max 100
    Image (898,-2 83x73), "HOME", image: VisuSymbols.Symbols.Home
        OnMouseClick:  Assign=HOME_1, Type=Assignment
    RoundedRectangle (895,429 48x34), "%1.2f", text variable: PLC_PRG_CFC_Davlenie_Stol_3_4.rCurrentValue
    RoundedRectangle (895,324 48x34), "%1.2f", text variable: PID_GLOBALS.g_rCurrentValue_Temperatura_Stol_3
    Lamp1 (950,315 24x23), variable: PLC_PRG_CFC_Temperatura_Stol_3.xMore, style: Lamp-Lamp1-Red
    Lamp1 (950,340 24x23), variable: PLC_PRG_CFC_Temperatura_Stol_3.xLess, style: Lamp-Lamp1-Blue
    Textfield (947,298 27x16), "ON"
    Textfield (947,365 27x16), "OFF"
    Textfield (947,405 27x16), "ON"
    Lamp1 (950,424 24x23), variable: PID_GLOBALS.xOut_More_Davlenie_Stol_3_4, style: Lamp-Lamp1-Blue
    Lamp1 (950,448 24x23), variable: PID_GLOBALS.xOut_Less_Davlenie_Stol_3_4, style: Lamp-Lamp1-Red
    Textfield (947,474 27x16), "OFF"
    Button (921,240 53x50), "?"
        OnMouseClick:  Assign=zapros, Type=Assignment
    Textfield (175,442 587x30), "МОДУЛЬ РАСШИРЕНИЯ В ОШИБКЕ!!!!!!!!!", invisible if: Connection.warning_1 = TRUE
    Image (138,0 659x554), invisible if: Connection.warning_1 = TRUE, image: VisuSymbols.Symbols.Caution
    Group (115,20 387x160), invisible if: PLC_PRG_archive.y1 = FALSE
        Rectangle (0,0 387x160), "Для того чтобы сохранить изменения нажмите да."
        Button (12,61 362x94), "ДА", invisible if: PLC_PRG_archive.y1 = FALSE
            tap PID_GLOBALS.yGO
            OnMouseClick: execute { PLC_PRG_archive.y1 := FALSE; }
END_VISUALIZATION

// Device/Application/Parostol_Zadanie/Zadanie_4
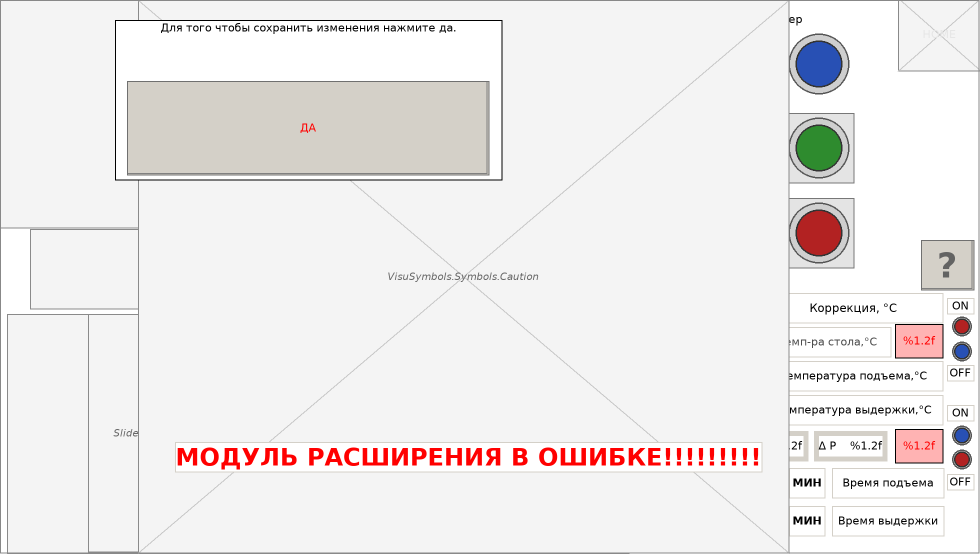
VISUALIZATION Zadanie_4  // 980x554
VAR_IN_OUT
END_VAR
VAR
	bResetTrigger : BOOL;
	bStart : BOOL;
	bStop : BOOL;
	bStore : BOOL;
	sStoreFilename : STRING;
	bRestore : BOOL;
	sRestoreFilename : STRING;
END_VAR
    Rectangle (3,-1 980x554)
    Histogram (7,314 622x240), scale format: %.1f, scale 0..100
        p518627256: °C
        p1518820177: PLC_PRG_Stol_4.arrHist1
        p102497268: PLC_PRG_Stol_4.arrHist1
        p788070771: ARRAY [0..3] OF REAL
    Slider (88,314 80x238), variable: PLC_PRG_Stol_4.Y1, scale 0..100
        OnValueChanged: execute { PLC_PRG_archive.z1 := TRUE; }
    Slider (215,313 80x238), variable: PLC_PRG_Stol_4.Y2, scale 0..100
        OnValueChanged: execute { PLC_PRG_archive.z1 := TRUE; }
    Slider (354,314 80x238), variable: PLC_PRG_Stol_4.Y3, scale 0..100
        OnValueChanged: execute { PLC_PRG_archive.z1 := TRUE; }
    Slider (487,314 80x238), variable: PLC_PRG_Stol_4.Y4, scale 0..100
        OnValueChanged: execute { PLC_PRG_archive.z1 := TRUE; }
    Trend (-3,-2 543x230)
        p758368661: dd.MM.yyyy
        p2423372160: H:mm:ss
        p2833066001: Visualization_Trend_Stol_4
        p2059293862: GenElemInst_240
    Line (925,485)
    Textfield (648,293 108x30)
        OnMouseClick: write the text variable via Default
    Textfield (648,395 108x30), "%d", text variable: PLC_PRG_Stol_4.Y3
        OnValueChanged: execute { PLC_PRG_archive.z1 := TRUE; }
        OnMouseClick: write the text variable via Default, min 0, max 100
    Textfield (648,327 108x30), "%d", text variable: PLC_PRG_Stol_4.Y1
        OnValueChanged: execute { PLC_PRG_archive.z1 := TRUE; }
        OnMouseClick: write the text variable via Default, min 0, max 100
    Textfield (649,468 50x30), "%d", text variable: PLC_PRG_Stol_4.HX2
        OnValueChanged: execute { PLC_PRG_archive.z1 := TRUE; }
        OnMouseClick: write the text variable via Default, min 0
    Textfield (764,293 179x30), "Коррекция, °C"
    Textfield (764,327 127x30), "Темп-ра стола,°C"
    Textfield (764,361 179x30), "Температура подъема,°C"
    Textfield (764,395 179x30), "Температура выдержки,°C"
    Textfield (832,468 112x30), "Время подъема"
    Textfield (649,507 50x30), "%d", text variable: PLC_PRG_Stol_4.HX3
        OnValueChanged: execute { PLC_PRG_archive.z1 := TRUE; }
        OnMouseClick: write the text variable via Default, min 0
    Textfield (832,506 112x30), "Время выдержки"
    Textfield (167,16 150x30), "%d °C, уставка", text variable: PID_GLOBALS.Temperatura_Stol_4_rSetPoint
    Textfield (734,468 50x30), "%d", text variable: PLC_PRG_Stol_4.MX2
        OnValueChanged: execute { PLC_PRG_archive.z1 := TRUE; }
        OnMouseClick: write the text variable via Default, min 0, max 59
    Textfield (704,468 25x30), "Ч"
    Textfield (789,468 36x30), "МИН"
    Textfield (734,507 50x30), "%d", text variable: PLC_PRG_Stol_4.MX3
        OnValueChanged: execute { PLC_PRG_archive.z1 := TRUE; }
        OnMouseClick: write the text variable via Default, min 0, max 59
    Textfield (704,507 25x30), "Ч"
    Textfield (789,506 36x30), "МИН"
    Checkbox (653,36 113x35), "Понедельник", variable: NVI_RETAIN.dateWeekStolThreeFour.9
        OnValueChanged: execute { PLC_PRG_archive.z1 := TRUE; }
    Checkbox (653,71 113x35), "Вторник", variable: NVI_RETAIN.dateWeekStolThreeFour.10
        OnValueChanged: execute { PLC_PRG_archive.z1 := TRUE; }
    Checkbox (653,106 113x35), "Среда", variable: NVI_RETAIN.dateWeekStolThreeFour.11
        OnValueChanged: execute { PLC_PRG_archive.z1 := TRUE; }
    Checkbox (653,141 113x35), "Четверг", variable: NVI_RETAIN.dateWeekStolThreeFour.12
        OnValueChanged: execute { PLC_PRG_archive.z1 := TRUE; }
    Checkbox (653,176 113x35), "Пятница", variable: NVI_RETAIN.dateWeekStolThreeFour.13
        OnValueChanged: execute { PLC_PRG_archive.z1 := TRUE; }
    Checkbox (653,211 113x35), "Суббота", variable: NVI_RETAIN.dateWeekStolThreeFour.14
        OnValueChanged: execute { PLC_PRG_archive.z1 := TRUE; }
    Checkbox (653,246 113x35), "Воскресенье", variable: NVI_RETAIN.dateWeekStolThreeFour.14
        OnValueChanged: execute { PLC_PRG_archive.z1 := TRUE; }
    Checkbox (653,2 237x35), "Активировать таймер", variable: NVI_RETAIN.dateWeekStolThreeFour.8
        OnValueChanged: execute { PLC_PRG_archive.z1 := TRUE; }
    Textfield (541,3 49x25), "Час"
    Textfield (598,3 49x25), "Мин"
    Textfield (541,38 49x30), "%d", text variable: NVI_RETAIN.hourMondayStolFour
        OnValueChanged: execute { PLC_PRG_archive.z1 := TRUE; }
        OnMouseClick: write the text variable via Default, min 0, max 23
    Textfield (598,38 49x30), "%d", text variable: NVI_RETAIN.minuteMondayStolFour
        OnValueChanged: execute { PLC_PRG_archive.z1 := TRUE; }
        OnMouseClick: write the text variable via Default, min 0, max 59
    Textfield (541,73 49x30), "%d", text variable: NVI_RETAIN.hourTuesdayStolFour
        OnValueChanged: execute { PLC_PRG_archive.z1 := TRUE; }
        OnMouseClick: write the text variable via Default, min 0, max 23
    Textfield (598,73 49x30), "%d", text variable: NVI_RETAIN.minuteTuesdayStolFour
        OnValueChanged: execute { PLC_PRG_archive.z1 := TRUE; }
        OnMouseClick: write the text variable via Default, min 0, max 59
    Textfield (541,108 49x30), "%d", text variable: NVI_RETAIN.hourWednesdayStolFour
        OnValueChanged: execute { PLC_PRG_archive.z1 := TRUE; }
        OnMouseClick: write the text variable via Default, min 0, max 23
    Textfield (541,143 49x30), "%d", text variable: NVI_RETAIN.hourThursdayStolFour
        OnValueChanged: execute { PLC_PRG_archive.z1 := TRUE; }
        OnMouseClick: write the text variable via Default, min 0, max 23
    Textfield (598,108 49x30), "%d", text variable: NVI_RETAIN.minuteWednesdayStolFour
        OnValueChanged: execute { PLC_PRG_archive.z1 := TRUE; }
        OnMouseClick: write the text variable via Default, min 0, max 59
    Textfield (541,213 49x30), "%d", text variable: NVI_RETAIN.hourSaturdayStolFour
        OnValueChanged: execute { PLC_PRG_archive.z1 := TRUE; }
        OnMouseClick: write the text variable via Default, min 0, max 23
    Textfield (598,178 49x30), "%d", text variable: NVI_RETAIN.minuteFridayStolFour
        OnValueChanged: execute { PLC_PRG_archive.z1 := TRUE; }
        OnMouseClick: write the text variable via Default, min 0, max 59
    Textfield (541,178 49x30), "%d", text variable: NVI_RETAIN.hourFridayStolFour
        OnValueChanged: execute { PLC_PRG_archive.z1 := TRUE; }
        OnMouseClick: write the text variable via Default, min 0, max 23
    Textfield (598,143 49x30), "%d", text variable: NVI_RETAIN.minuteThursdayStolFour
        OnValueChanged: execute { PLC_PRG_archive.z1 := TRUE; }
        OnMouseClick: write the text variable via Default, min 0, max 59
    Textfield (541,248 49x30), "%d", text variable: NVI_RETAIN.hourSundayStolFour
        OnValueChanged: execute { PLC_PRG_archive.z1 := TRUE; }
        OnMouseClick: write the text variable via Default, min 0, max 23
    Textfield (598,213 49x30), "%d", text variable: NVI_RETAIN.minuteSaturdayStolFour
        OnValueChanged: execute { PLC_PRG_archive.z1 := TRUE; }
        OnMouseClick: write the text variable via Default, min 0, max 59
    Textfield (598,248 49x30), "%d", text variable: NVI_RETAIN.minuteSundayStolFour
        OnValueChanged: execute { PLC_PRG_archive.z1 := TRUE; }
        OnMouseClick: write the text variable via Default, min 0, max 59
    PushSwitch (784,113 70x70), variable: PLC_PRG_Stol_4.START, behaviour: TAP, style: Switch-PushSwitch-Green
    Lamp1 (784,29 70x70), variable: PLC_PRG_Stol_4.INDIKATOR, style: Lamp-Lamp1-Blue
    PushSwitch (784,198 70x70), variable: PLC_PRG_Stol_4.STOP, behaviour: TAP, style: Switch-PushSwitch-Red
    Textfield (1314,316 0x1)
    Textfield (860,49 84x30), "РАБОТА"
    Textfield (860,133 94x30), "СТАРТ РУЧН."
    Textfield (860,218 84x30), "СТОП"
    DateRangeSelector (30,229 509x80)
        p758368661: dd.MM
        p2423372160: H:mm
        p1661464551: GenElemInst_30
    Textfield (648,431 76x30), "Pобр. %1.2f", text variable: PID_GLOBALS.g_rCurrentValue_Davlenie_Podacha_Stol_3_4
    Textfield (730,431 78x30), "Pпод. %1.2f", text variable: PID_GLOBALS.g_rCurrentValue_Davlenie_Obratnaja_Stol_3_4
        OnMouseClick: write the text variable via Default, min 0, max 100
    Textfield (814,431 73x30), "Δ Р %1.2f", text variable: PLC_PRG_CFC_Davlenie_Stol_3_4.Davlenie_Stol_3_4_rSetPoint
        OnValueChanged: execute { PLC_PRG_archive.z1 := TRUE; }
        OnMouseClick: write the text variable via Default, min 0, max 100
    Textfield (168,163 220x38), "Термостол №4"
    Textfield (648,361 108x30), "%d", text variable: PLC_PRG_Stol_4.Y2
        OnValueChanged: execute { PLC_PRG_archive.z1 := TRUE; }
        OnMouseClick: write the text variable via Default, min 0, max 100
    Image (898,-2 83x73), "HOME", image: VisuSymbols.Symbols.Home
        OnMouseClick:  Assign=HOME_1, Type=Assignment
    RoundedRectangle (895,429 48x34), "%1.2f", text variable: PLC_PRG_CFC_Davlenie_Stol_3_4.rCurrentValue
    RoundedRectangle (895,324 48x34), "%1.2f", text variable: PID_GLOBALS.g_rCurrentValue_Temperatura_Stol_4
    Textfield (947,474 27x16), "OFF"
    Lamp1 (950,448 24x23), variable: PID_GLOBALS.xOut_Less_Davlenie_Stol_3_4, style: Lamp-Lamp1-Red
    Lamp1 (950,424 24x23), variable: PID_GLOBALS.xOut_More_Davlenie_Stol_3_4, style: Lamp-Lamp1-Blue
    Textfield (947,405 27x16), "ON"
    Textfield (947,365 27x16), "OFF"
    Lamp1 (950,340 24x23), variable: PLC_PRG_CFC_Temperatura_Stol_4.xLess, style: Lamp-Lamp1-Blue
    Lamp1 (950,315 24x23), variable: PLC_PRG_CFC_Temperatura_Stol_4.xMore, style: Lamp-Lamp1-Red
    Textfield (947,298 27x16), "ON"
    Button (921,240 53x50), "?"
        OnMouseClick:  Assign=zapros, Type=Assignment
    Image (138,0 651x553), invisible if: Connection.warning_1 = TRUE, image: VisuSymbols.Symbols.Caution
    Textfield (175,442 587x30), "МОДУЛЬ РАСШИРЕНИЯ В ОШИБКЕ!!!!!!!!!", invisible if: Connection.warning_1 = TRUE
    Group (115,20 387x160), invisible if: PLC_PRG_archive.z1 = FALSE
        Rectangle (0,0 387x160), "Для того чтобы сохранить изменения нажмите да."
        Button (12,61 362x94), "ДА", invisible if: PLC_PRG_archive.z1 = FALSE
            tap PID_GLOBALS.yGO
            OnMouseClick: execute { PLC_PRG_archive.z1 := FALSE; }
END_VISUALIZATION

// Device/Application/Parostol_Zadanie/Visualization_CFC_Temperatura_4
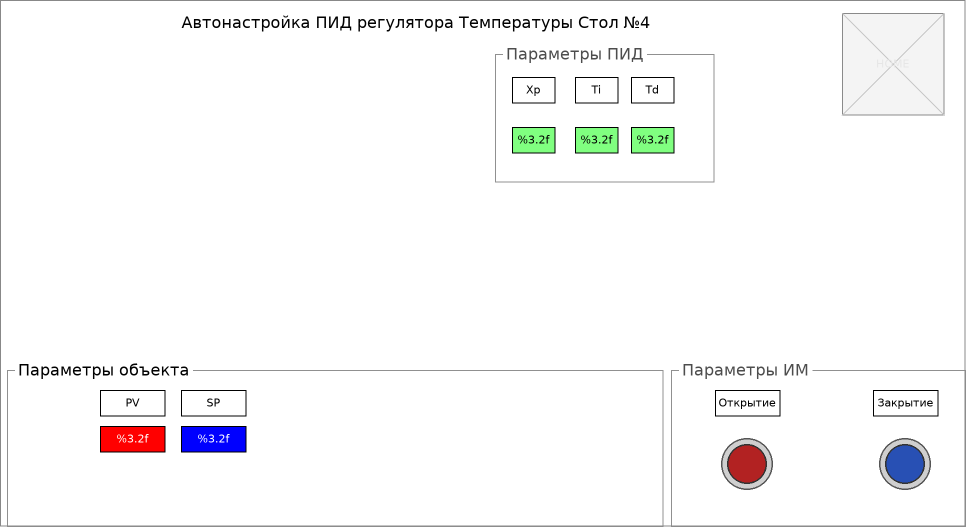
VISUALIZATION Visualization_CFC_Temperatura_4  // 966x527
    GroupBox (7,362 656x165), "Параметры объекта"
        RoundedRectangle (93,64 65x26), "%3.2f", text variable: PID_GLOBALS.g_rCurrentValue_Temperatura_Stol_4
    GroupBox (495,46 219x136), "Параметры ПИД"
        RoundedRectangle (136,81 43x26), "%3.2f", text variable: PLC_PRG_CFC_Temperatura_Stol_4.rTd
            OnMouseClick: write the text variable via Default
        RoundedRectangle (80,81 43x26), "%3.2f", text variable: PLC_PRG_CFC_Temperatura_Stol_4.rTi
            OnMouseClick: write the text variable via Default
        RoundedRectangle (17,81 43x26), "%3.2f", text variable: PLC_PRG_CFC_Temperatura_Stol_4.rXp
            OnMouseClick: write the text variable via Default
        Rectangle (17,31 43x26), "Xp"
        Rectangle (80,31 43x26), "Ti"
        Rectangle (136,31 43x26), "Td"
    RoundedRectangle (181,426 65x26), "%3.2f", text variable: PLC_PRG_Stol_4.Y1
        OnMouseClick: write the text variable via Default
    Rectangle (100,390 65x26), "PV", tooltip "Значение температуры"
    Rectangle (181,390 65x26), "SP", tooltip "Уставка температуры"
    GroupBox (671,362 295x165), "Параметры ИМ"
        Rectangle (44,28 65x26), "Открытие"
        Rectangle (202,28 65x26), "Закрытие"
        Lamp1 (46,72 60x60), variable: PLC_PRG_CFC_Temperatura_Stol_4.xMore, style: Lamp-Lamp1-Red
        Lamp1 (204,72 60x60), variable: PLC_PRG_CFC_Temperatura_Stol_4.xLess, style: Lamp-Lamp1-Blue
    Image (842,13 102x102), "HOME", image: VisuSymbols.Symbols.Home
        OnMouseClick:  Assign=HOME_1, Type=Assignment
    Rectangle (107,7 618x31), "Автонастройка ПИД регулятора Температуры Стол №4"
END_VISUALIZATION

// Device/Application/Parostol_Zadanie/Visualization_CFC_Temperatura_2
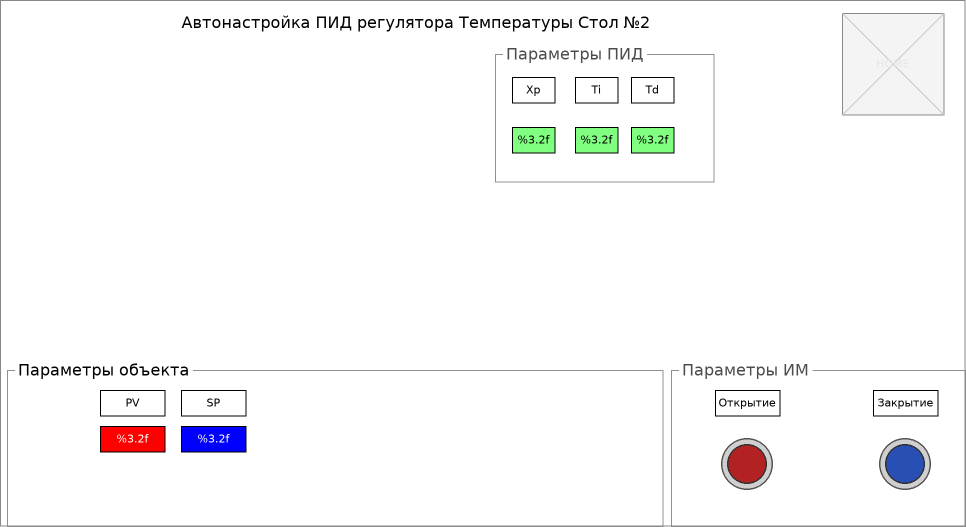
VISUALIZATION Visualization_CFC_Temperatura_2  // 966x527
    GroupBox (7,362 656x165), "Параметры объекта"
        RoundedRectangle (93,64 65x26), "%3.2f", text variable: PID_GLOBALS.g_rCurrentValue_Temperatura_Stol_2
    GroupBox (495,46 219x136), "Параметры ПИД"
        RoundedRectangle (136,81 43x26), "%3.2f", text variable: PLC_PRG_CFC_Temperatura_Stol_2.rTd
            OnMouseClick: write the text variable via Default
        RoundedRectangle (80,81 43x26), "%3.2f", text variable: PLC_PRG_CFC_Temperatura_Stol_2.rTi
            OnMouseClick: write the text variable via Default
        RoundedRectangle (17,81 43x26), "%3.2f", text variable: PLC_PRG_CFC_Temperatura_Stol_2.rXp
            OnMouseClick: write the text variable via Default
        Rectangle (17,31 43x26), "Xp"
        Rectangle (80,31 43x26), "Ti"
        Rectangle (136,31 43x26), "Td"
    RoundedRectangle (181,426 65x26), "%3.2f", text variable: PLC_PRG_Stol_2.Y1
        OnMouseClick: write the text variable via Default
    Rectangle (100,390 65x26), "PV", tooltip "Значение температуры"
    Rectangle (181,390 65x26), "SP", tooltip "Уставка температуры"
    GroupBox (671,362 295x165), "Параметры ИМ"
        Rectangle (44,28 65x26), "Открытие"
        Rectangle (202,28 65x26), "Закрытие"
        Lamp1 (46,72 60x60), variable: PLC_PRG_CFC_Temperatura_Stol_2.xMore, style: Lamp-Lamp1-Red
        Lamp1 (204,72 60x60), variable: PLC_PRG_CFC_Temperatura_Stol_2.xLess, style: Lamp-Lamp1-Blue
    Image (842,13 102x102), "HOME", image: VisuSymbols.Symbols.Home
        OnMouseClick:  Assign=HOME_1, Type=Assignment
    Rectangle (107,7 618x31), "Автонастройка ПИД регулятора Температуры Стол №2"
END_VISUALIZATION

// Device/Application/Parostol_Zadanie/Visualization_CFC_Temperatura_3
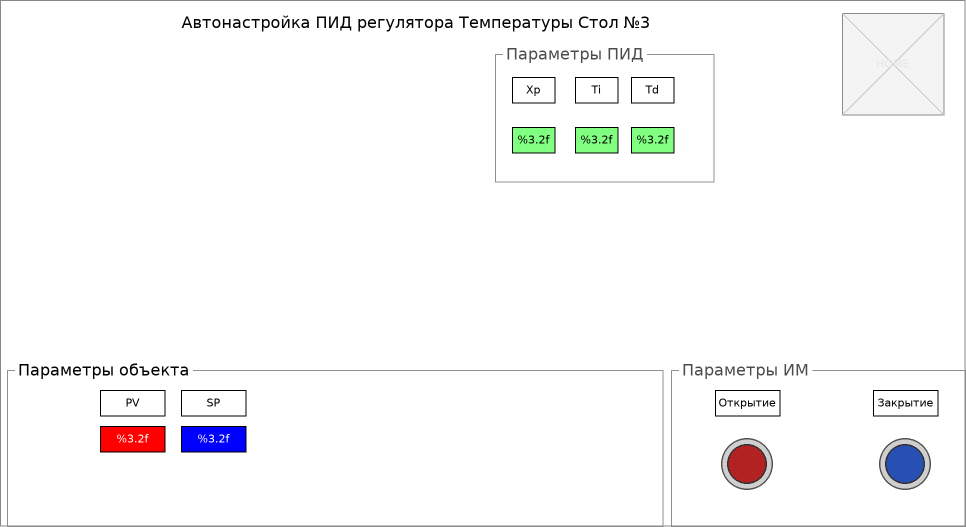
VISUALIZATION Visualization_CFC_Temperatura_3  // 966x527
    GroupBox (7,362 656x165), "Параметры объекта"
        RoundedRectangle (93,64 65x26), "%3.2f", text variable: PID_GLOBALS.g_rCurrentValue_Temperatura_Stol_3
    GroupBox (495,46 219x136), "Параметры ПИД"
        RoundedRectangle (136,81 43x26), "%3.2f", text variable: PLC_PRG_CFC_Temperatura_Stol_3.rTd
            OnMouseClick: write the text variable via Default
        RoundedRectangle (80,81 43x26), "%3.2f", text variable: PLC_PRG_CFC_Temperatura_Stol_3.rTi
            OnMouseClick: write the text variable via Default
        RoundedRectangle (17,81 43x26), "%3.2f", text variable: PLC_PRG_CFC_Temperatura_Stol_3.rXp
            OnMouseClick: write the text variable via Default
        Rectangle (17,31 43x26), "Xp"
        Rectangle (80,31 43x26), "Ti"
        Rectangle (136,31 43x26), "Td"
    RoundedRectangle (181,426 65x26), "%3.2f", text variable: PLC_PRG_Stol_3.Y1
        OnMouseClick: write the text variable via Default
    Rectangle (100,390 65x26), "PV", tooltip "Значение температуры"
    Rectangle (181,390 65x26), "SP", tooltip "Уставка температуры"
    GroupBox (671,362 295x165), "Параметры ИМ"
        Rectangle (44,28 65x26), "Открытие"
        Rectangle (202,28 65x26), "Закрытие"
        Lamp1 (46,72 60x60), variable: PLC_PRG_CFC_Temperatura_Stol_3.xMore, style: Lamp-Lamp1-Red
        Lamp1 (204,72 60x60), variable: PLC_PRG_CFC_Temperatura_Stol_3.xLess, style: Lamp-Lamp1-Blue
    Image (842,13 102x102), "HOME", image: VisuSymbols.Symbols.Home
        OnMouseClick:  Assign=HOME_1, Type=Assignment
    Rectangle (107,7 618x31), "Автонастройка ПИД регулятора Температуры Стол №3"
END_VISUALIZATION

// Device/Application/instructions/HELP
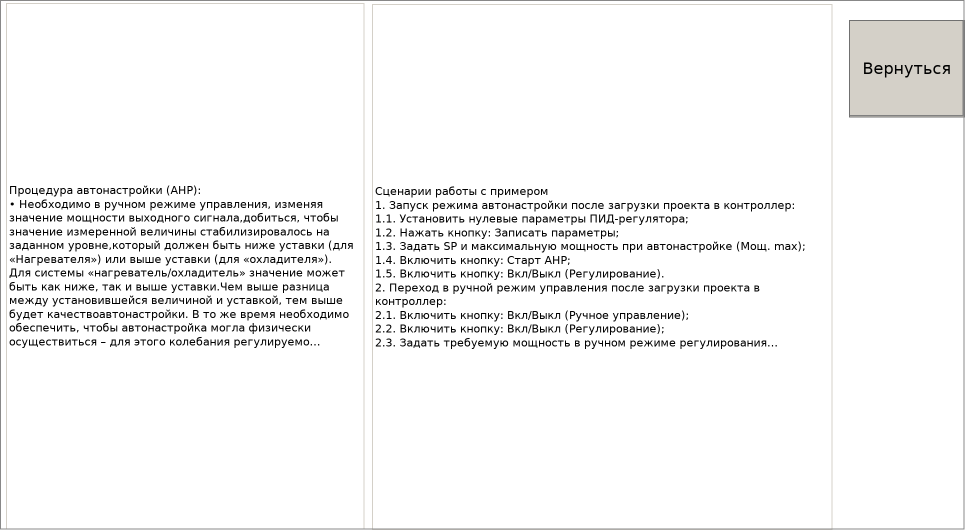
VISUALIZATION HELP  // 965x530
    Textfield (6,3 358x526), "Процедура автонастройки (АНР): • Необходимо в ручном режиме управления, изменяя значение мощности выходного сигнала,добиться, чтобы значение измеренной величины стабилизировалось на заданном уровне,который должен быть ниже уставки (для «Нагревателя») или выше уставки (для «охладителя»). Для системы «нагреватель/охладитель» значение может быть как ниже, так и выше уставки.Чем выше разница между установившейся величиной и уставкой, тем выше будет качествоавтонастройки. В то же время необходимо обеспечить, чтобы автонастройка могла физически осуществиться – для этого колебания регулируемой величины в диапазоне [Уставка АНР -зона колебаний АНР...Уставка АНР + зона колебаний АНР] должны быть достижимы при изменении выходного сигнала. Также, очевидно, такие колебания не должны приводить к негативным воздействиям на объект регулирования. • Выключить в программе ФБ ПИД-регулятора и выполнить его сброс присвоив экземпляру ФБ ПИД-регулятора пустой (не вызываемый в программе) экземпляр аналогичного ПИДрегулятора, так как при проведении автонастройки память ФБ должны быть очищена. • Режим автонастройки запускается только из режима регулирования, поэтому необходимо записать нулевые (какие-либо) коэффициенты ПИД-регулятора (перейти в режим START_PID); • Включить в программе ФБ ПИД-регулятора таким образом, чтобы в первом цикле контроллера ФБ ПИД регулятора перешел в режим регулирования со всеми установленными параметрами, кроме SP, чтобы не началась выработка регулирующих воздействий. Также необходимо предусмотреть, чтобы во втором цикле контроллера произошел автоматический пуск автонастройки одновременно с записью уставки регулятора."
    Button (849,20 116x97), "Вернуться"
        OnMouseClick:  Type=Previous
    Textfield (372,4 460x526), "Сценарии работы с примером 1. Запуск режима автонастройки после загрузки проекта в контроллер: 1.1. Установить нулевые параметры ПИД-регулятора; 1.2. Нажать кнопку: Записать параметры; 1.3. Задать SP и максимальную мощность при автонастройке (Мощ. max); 1.4. Включить кнопку: Старт АНР; 1.5. Включить кнопку: Вкл/Выкл (Регулирование). 2. Переход в ручной режим управления после загрузки проекта в контроллер: 2.1. Включить кнопку: Вкл/Выкл (Ручное управление); 2.2. Включить кнопку: Вкл/Выкл (Регулирование); 2.3. Задать требуемую мощность в ручном режиме регулирования; 2.4. Нажать кнопку: Запись. 3. Выход из ручного режима работы: 3.1. Выключить кнопку: Вкл/Выкл (Регулирование); 3.2. Выключить кнопку: Вкл/Выкл (Ручное управление); 4. Запуск режима автонастройки после выхода из ручного режима работы: 4.1. Нажать кнопку: Сброс ПИД; 4.2. Установить нулевые параметры ПИД-регулятора; 4.3. Нажать кнопку: Записать параметры; 4.4. Задать SP и Максимальную мощность при автонастройке (Мощ. max); 4.5. Включить кнопку: Старт АНР; 4.6. Включить кнопку: Вкл/Выкл (Регулирование). 5. Запуск режима регулирования после загрузки проекта в контроллер: 5.1. Установить параметры ПИД-регулятора; 5.2. Нажать кнопку: Записать параметры; 5.3. Задать SP; 5.4. Нажать кнопку: Записать SP; 5.5. Включить кнопку: Вкл/Выкл (Регулирование). 6. Запуск режима регулирования при выходе из ручного режима работы: 6.1. Установить параметры ПИД-регулятора; 6.2. Нажать кнопку: Записать параметры; Выключить кнопку: Вкл/Выкл (Ручное управление)."
END_VISUALIZATION

// Device/Application/Parostol_Zadanie/Visualization_CFC_Davlenie_3_4
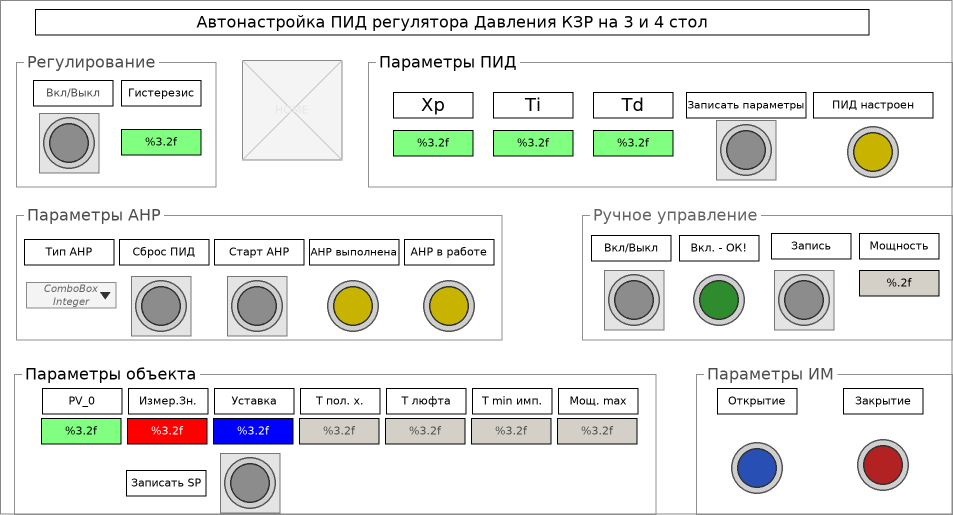
VISUALIZATION Visualization_CFC_Davlenie_3_4  // 953x515
    GroupBox (16,207 486x133), "Параметры АНР"
        Rectangle (293,32 90x26), "АНР выполнена"
        Lamp1 (307,69 60x60), variable: PLC_PRG_CFC_Davlenie_Stol_3_4.xAutotuneCompleted, style: Lamp-Lamp1-Yellow
        Rectangle (103,32 90x26), "Сброс ПИД"
        PushSwitchLed (211,69 60x60), variable: PLC_PRG_CFC_Davlenie_Stol_3_4.xStartAutotune, behaviour: TOGGLE, style: Switch-PushSwitchLed-Gray
        PushSwitch (115,69 60x60), variable: PLC_PRG_CFC_Davlenie_Stol_3_4.xReset, behaviour: TAP, style: Switch-PushSwitch-Gray
        Rectangle (388,32 90x26), "АНР в работе"
        Lamp1 (403,69 60x60), variable: PLC_PRG_CFC_Davlenie_Stol_3_4.xAutotuneInProgress, style: Lamp-Lamp1-Yellow
        Rectangle (198,32 90x26), "Старт АНР"
        ComboBoxInteger (10,75 90x26), variable: PLC_PRG_CFC_Davlenie_Stol_3_4.eAutotuneMode, text list: 'ANR_MODE'
    Rectangle (24,239 90x26), "Тип АНР"
    GroupBox (16,54 200x133), "Регулирование"
        PushSwitchLed (23,59 60x60), variable: PLC_PRG_CFC_Davlenie_Stol_3_4.xIsEnabledPid, behaviour: TOGGLE, style: Switch-PushSwitchLed-Gray
        Rectangle (105,26 80x26), "Гистерезис"
        RoundedRectangle (105,75 80x26), "%3.2f", text variable: PLC_PRG_CFC_Davlenie_Stol_3_4.rDeadBand
            OnMouseClick: write the text variable via Default
    Rectangle (33,80 80x26), "Вкл/Выкл"
    GroupBox (368,54 585x133), "Параметры ПИД"
        Lamp1 (475,68 60x60), variable: PLC_PRG_CFC_Davlenie_Stol_3_4.xIsPidValidSettings, style: Lamp-Lamp1-Yellow
        PushSwitch (348,66 60x60), variable: PLC_PRG_CFC_Davlenie_Stol_3_4.xWritePidSettings, behaviour: TAP, style: Switch-PushSwitch-Gray
        Rectangle (318,38 120x26), "Записать параметры"
        Rectangle (445,38 120x26), "ПИД настроен"
    RoundedRectangle (393,130 80x26), "%3.2f", text variable: PLC_PRG_CFC_Davlenie_Stol_3_4.rXp
        OnMouseClick: write the text variable via Default
    RoundedRectangle (493,130 80x26), "%3.2f", text variable: PLC_PRG_CFC_Davlenie_Stol_3_4.rTi
        OnMouseClick: write the text variable via Default
    RoundedRectangle (593,130 80x26), "%3.2f", text variable: PLC_PRG_CFC_Davlenie_Stol_3_4.rTd
        OnMouseClick: write the text variable via Default
    Rectangle (393,92 80x26), "Xp"
    Rectangle (493,92 80x26), "Ti"
    Rectangle (593,92 80x26), "Td"
    GroupBox (696,366 257x149), "Параметры ИМ"
        Rectangle (21,22 80x26), "Открытие"
        Rectangle (147,22 80x26), "Закрытие"
        Lamp1 (31,72 60x60), variable: PID_GLOBALS.xOut_More_Davlenie_Stol_3_4, style: Lamp-Lamp1-Blue
        Lamp1 (157,69 60x60), variable: PID_GLOBALS.xOut_Less_Davlenie_Stol_3_4, style: Lamp-Lamp1-Red
    GroupBox (14,366 642x149), "Параметры объекта"
        RoundedRectangle (113,52 80x26), "%3.2f", text variable: PLC_PRG_CFC_Davlenie_Stol_3_4.rCurrentValue
        RoundedRectangle (371,52 80x26), "%3.2f", text variable: PLC_PRG_CFC_Davlenie_Stol_3_4.rTluft
            OnMouseClick: write the text variable via Default
        RoundedRectangle (543,52 80x26), "%3.2f", text variable: PLC_PRG_CFC_Davlenie_Stol_3_4.rDy_anr
            OnMouseClick: write the text variable via Default
        PushSwitch (206,87 60x60), variable: PLC_PRG_CFC_Davlenie_Stol_3_4.xSetSP, behaviour: TAP, style: Switch-PushSwitch-Gray
        Rectangle (112,104 80x26), "Записать SP"
        Rectangle (200,22 80x26), "Уставка", tooltip "Уставка давления"
        RoundedRectangle (199,52 80x26), "%3.2f", text variable: PLC_PRG_CFC_Davlenie_Stol_3_4.Davlenie_Stol_3_4_rSetPoint
            OnMouseClick: write the text variable via Default
        RoundedRectangle (457,52 80x26), "%3.2f", text variable: PLC_PRG_CFC_Davlenie_Stol_3_4.rTimp
            OnMouseClick: write the text variable via Default
        RoundedRectangle (285,52 80x26), "%3.2f", text variable: PLC_PRG_CFC_Davlenie_Stol_3_4.rTval
            OnMouseClick: write the text variable via Default
    RoundedRectangle (41,418 80x26), "%3.2f", text variable: PLC_PRG_CFC_Davlenie_Stol_3_4.rSteadyValue
        OnMouseClick: write the text variable via Default
    Rectangle (42,388 80x26), "PV_0", tooltip "Значение регулируемого параметра при нулевом уровне мощности (при Y=0)"
    Rectangle (128,388 80x26), "Измер.Зн.", tooltip "Значение давления"
    Rectangle (300,388 80x26), "Т пол. х.", tooltip "Время полного хода ИМ, сек."
    Rectangle (386,388 80x26), "Т люфта", tooltip "Время выборки люфта ИМ, сек."
    Rectangle (472,388 80x26), "Т min имп.", tooltip "Минимальная длительность импульса, сек."
    Rectangle (558,388 80x26), "Мощ. max", tooltip "Размах мощности (в процентах), выдаваемый на задвижку от текущей позиции при АНР. Например, при положении задвижки 50% и значении DY_ANR=25% в ходе АНР задвижка будет перемещаться от 25 до 75% (без учета влияния физических процессов на перемещение задвижки) Диапазон возможныз значений: 0.0...100.0 (%)"
    GroupBox (582,207 371x133), "Ручное управление"
        PushSwitchLed (22,63 60x60), variable: PLC_PRG_CFC_Davlenie_Stol_3_4.xManualMode, behaviour: TOGGLE, style: Switch-PushSwitchLed-Gray
        PushSwitch (192,63 60x60), variable: PLC_PRG_CFC_Davlenie_Stol_3_4.xManual_set, behaviour: TAP, style: Switch-PushSwitch-Gray
        Rectangle (189,26 80x26), "Запись"
        RoundedRectangle (277,63 80x26), "%.2f", text variable: PLC_PRG_CFC_Davlenie_Stol_3_4.rManual_mean
            OnMouseClick: write the text variable via Default
        Rectangle (277,26 80x26), "Мощность"
        Lamp1 (107,63 60x60), variable: PLC_PRG_CFC_Davlenie_Stol_3_4.xSetManualOK, style: Lamp-Lamp1-Green
        Rectangle (9,28 80x26), "Вкл/Выкл"
        Rectangle (97,28 80x26), "Вкл. - ОК!"
    Rectangle (35,9 834x26), "Автонастройка ПИД регулятора Давления КЗР на 3 и 4 стол"
    Image (242,60 100x100), "HOME", image: VisuSymbols.Symbols.Home
        OnMouseClick:  Assign=HOME_1, Type=Assignment
END_VISUALIZATION

// Device/Application/instructions/zapros
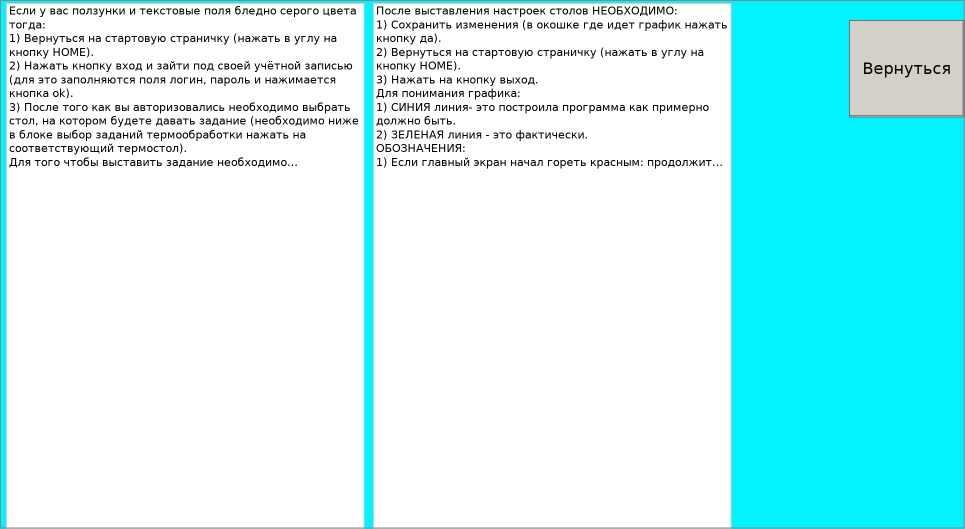
VISUALIZATION zapros  // 965x529
    Textfield (6,3 358x526), "Если у вас ползунки и текстовые поля бледно серого цвета тогда: 1) Вернуться на стартовую страничку (нажать в углу на кнопку HOME). 2) Нажать кнопку вход и зайти под своей учётной записью (для это заполняются поля логин, пароль и нажимается кнопка ok). 3) После того как вы авторизовались необходимо выбрать стол, на котором будете давать задание (необходимо ниже в блоке выбор заданий термообработки нажать на соответствующий термостол). Для того чтобы выставить задание необходимо: 1) Выставить температуру стола (Темп-ра стола,°C) (Температуру стола можно померить прибором и для сверки посмотреть температуру рядом в красном поле). 2) Выставить температуру подъема стола (Температура подъема,°C). 3) Выставить температуру выдержки стола (Температура выдержки,°C). 4) Выставить Δ Р (Давление). 5) Выставить время подъема (Через данный промежуток времени температура стола будет равняться значению, которое вы выставили выше). 6) Выставить время выдержки (Время, которое стол будет поддерживать температуру выдержки, заданную выше). 7) Сверху выбрать день недели (Поставить галочку на соответствующем поле) и настроить время для начала работы (во сколько начнется). 8) Еще выше ОБЯЗАТЕЛЬНО поставить галочку АКТИВИРОВАТЬ ТАЙМЕР."
    Button (849,20 116x97), "Вернуться"
        OnMouseClick:  Type=Previous
    Textfield (373,3 358x526), "После выставления настроек столов НЕОБХОДИМО: 1) Сохранить изменения (в окошке где идет график нажать кнопку да). 2) Вернуться на стартовую страничку (нажать в углу на кнопку HOME). 3) Нажать на кнопку выход. Для понимания графика: 1) СИНИЯ линия- это построила программа как примерно должно быть. 2) ЗЕЛЕНАЯ линия - это фактически. ОБОЗНАЧЕНИЯ: 1) Если главный экран начал гореть красным: продолжить работу и сообщить об этом в отдел КИПиА. 2) Если при заходе на нужный термостол горит ошибка “Модуль расширения в ошибке” сообщить об этом в отдел КИПиА."
END_VISUALIZATION

// Device/Application/instructions/instrykcai_avtoriz
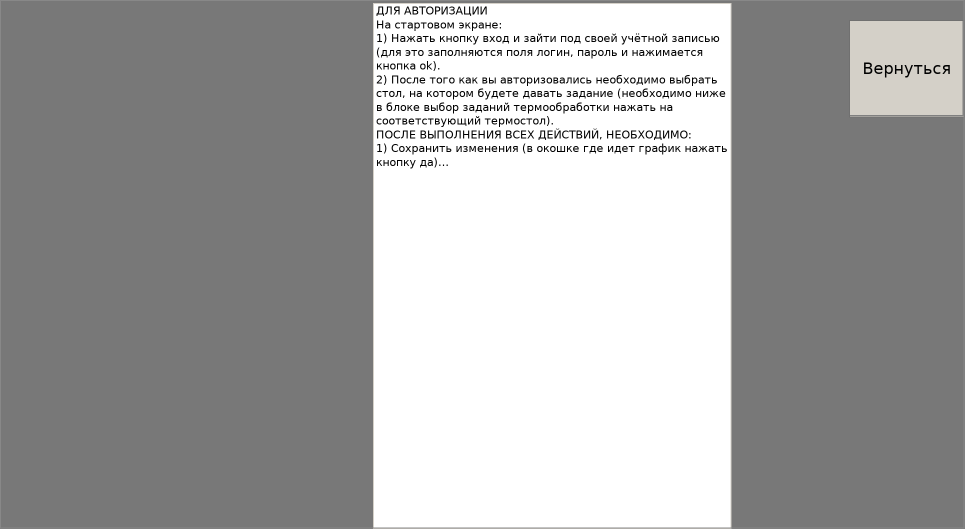
VISUALIZATION instrykcai_avtoriz  // 965x529
    Button (849,20 116x97), "Вернуться"
        OnMouseClick:  Type=Previous
    Textfield (373,3 358x526), "ДЛЯ АВТОРИЗАЦИИ На стартовом экране: 1) Нажать кнопку вход и зайти под своей учётной записью (для это заполняются поля логин, пароль и нажимается кнопка ok). 2) После того как вы авторизовались необходимо выбрать стол, на котором будете давать задание (необходимо ниже в блоке выбор заданий термообработки нажать на соответствующий термостол). ПОСЛЕ ВЫПОЛНЕНИЯ ВСЕХ ДЕЙСТВИЙ, НЕОБХОДИМО: 1) Сохранить изменения (в окошке где идет график нажать кнопку да). 2) Вернуться на стартовую страничку (нажать в углу на кнопку HOME). 3) Нажать на кнопку выход. ОБОЗНАЧЕНИЯ: 1) Если главный экран начал гореть красным: продолжить работу и сообщить об этом в отдел КИПиА. 2) Если при заходе на нужный термостол горит ошибка “Модуль расширения в ошибке” сообщить об этом в отдел КИПиА."
END_VISUALIZATION

(* text list System (id | default)
  Apr | Apr
  April | April
  Aug | Aug
  August | August
  Dec | Dec
  December | December
  Feb | Feb
  February | February
  Fri | Fri
  Friday | Friday
  Jan | Jan
  January | January
  Jul | Jul
  July | July
  Jun | Jun
  June | June
  Mar | Mar
  March | March
  May | May
  May_3Letter | May
  Mon | Mon
  Monday | Monday
  Nov | Nov
  November | November
  Oct | Oct
  October | October
  Sat | Sat
  Saturday | Saturday
  Sep | Sep
  September | September
  Sun | Sun
  Sunday | Sunday
  Thu | Thu
  Thursday | Thursday
  Tue | Tue
  Tuesday | Tuesday
  Wed | Wed
  Wednesday | Wednesday
   |  *)

(* text list ANR_MODE (id | default)
  0 | Динамическая
  1 | Плавная
   |  *)

(* text list ANR_WAVE_COUNT (id | default)
  0 | Одна волна
  1 | Две волны
   |  *)

(* text list ERROR_PID (id | default)
  0 | Нет ошибок
  1 | Некорректное PV
  2 | Ошибка обратной связи
   |  *)

(* text list STATE_PID (id | default)
  0 | Первый запуск
  1 | Инициализация регулятора
  2 | Запуск АНР
  3 | АНР в процессе
  4 | ПИД запущен
  5 | ПИД в работе
  6 | Ручной режим
   |  *)
